KUKA KRL program: MyProgram_177().src

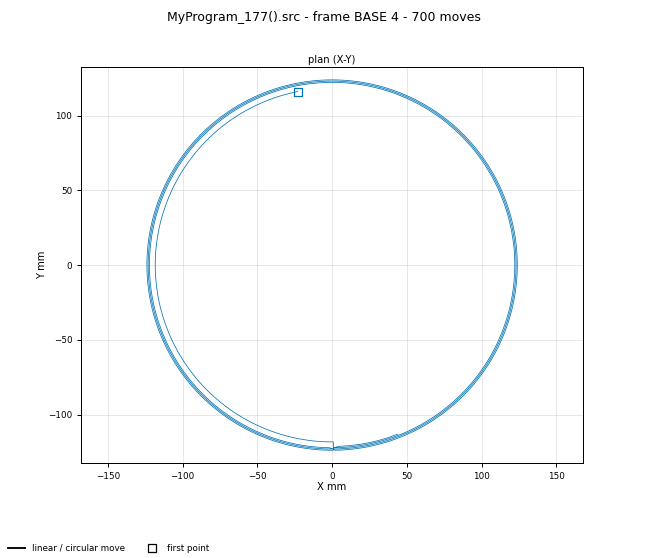
[picture p0: tool path of MyProgram_177().src in frame BASE 4, 700 of 700 moves have a stored position in this frame; points joined in program order, loops and branches not executed]
&ACCESS RVP
&REL 1
&PARAM TEMPLATE = C:\KRC\Roboter\Template\vorgabe
&PARAM EDITMASK = *
DEF MyProgram_177()
; ---- Setting reference (Base) ----
$BASE = BASE_DATA[4]

; --------------------------
; ---- Setting tool (TCP) ----
$TOOL = TOOL_DATA[3]
; --------------------------

$VEL.CP = VEL_APROX_PRINT
Startdeposition()
$VEL.CP = VEL_PRINT
LIN {X -23.0554,Y 116.0381,Z 130,A 97.2473,B 24.9369,C -1.8336,E1 24.968,E2 348.7277} C_DIS
LIN {X -25.5832,Y 115.5056,Z 130,A 98.5297,B 24.9369,C -1.8339,E1 24.9645,E2 347.4431} C_DIS
LIN {X -28.4099,Y 114.843,Z 130,A 99.9093,B 24.9371,C -1.8314,E1 24.9608,E2 346.0675} C_DIS
LIN {X -31.5451,Y 114.0233,Z 130,A 101.4825,B 24.9372,C -1.8299,E1 24.9566,E2 344.4954} C_DIS
LIN {X -33.9988,Y 113.3142,Z 130,A 102.7524,B 24.9372,C -1.8299,E1 24.9532,E2 343.2232} C_DIS
LIN {X -38.179,Y 111.9751,Z 130,A 104.8537,B 24.9375,C -1.8263,E1 24.9476,E2 341.1266} C_DIS
LIN {X -41.2308,Y 110.8892,Z 130,A 106.4224,B 24.9376,C -1.8243,E1 24.9435,E2 339.5598} C_DIS
LIN {X -43.9338,Y 109.8464,Z 130,A 107.833,B 24.9377,C -1.8227,E1 24.9398,E2 338.1499} C_DIS
LIN {X -46.5663,Y 108.7563,Z 130,A 109.2196,B 24.9378,C -1.8209,E1 24.9363,E2 336.7642} C_DIS
LIN {X -48.9465,Y 107.7046,Z 130,A 110.5124,B 24.9378,C -1.8205,E1 24.933,E2 335.4694} C_DIS
LIN {X -51.8783,Y 106.3252,Z 130,A 112.0577,B 24.9381,C -1.8169,E1 24.9291,E2 333.9286} C_DIS
LIN {X -54.4655,Y 105.0233,Z 130,A 113.4668,B 24.9383,C -1.8149,E1 24.9256,E2 332.5205} C_DIS
LIN {X -56.7349,Y 103.8132,Z 130,A 114.744,B 24.9383,C -1.8141,E1 24.9224,E2 331.2415} C_DIS
LIN {X -59.5311,Y 102.237,Z 130,A 116.2695,B 24.9386,C -1.81,E1 24.9188,E2 329.7212} C_DIS
LIN {X -61.9831,Y 100.769,Z 130,A 117.6521,B 24.9388,C -1.8074,E1 24.9155,E2 328.3406} C_DIS
LIN {X -64.0841,Y 99.4443,Z 130,A 118.8954,B 24.9388,C -1.8069,E1 24.9125,E2 327.0945} C_DIS
LIN {X -66.9275,Y 97.5557,Z 130,A 120.5341,B 24.9391,C -1.8029,E1 24.9087,E2 325.4598} C_DIS
LIN {X -69.0267,Y 96.0799,Z 130,A 121.7828,B 24.9392,C -1.8006,E1 24.9059,E2 324.2122} C_DIS
LIN {X -71.633,Y 94.1548,Z 130,A 123.5319,B 24.9389,C -1.805,E1 24.902,E2 322.4465} C_DIS
LIN {X -74.471,Y 91.9237,Z 130,A 125.1574,B 24.9395,C -1.7959,E1 24.8985,E2 320.8364} C_DIS
LIN {X -77.1406,Y 89.6968,Z 130,A 126.8154,B 24.9399,C -1.791,E1 24.8949,E2 319.1838} C_DIS
LIN {X -79.8507,Y 87.2914,Z 130,A 128.6126,B 24.94,C -1.7887,E1 24.8912,E2 317.3847} C_DIS
LIN {X -82.1926,Y 85.0898,Z 130,A 130.1847,B 24.9402,C -1.7857,E1 24.888,E2 315.8135} C_DIS
LIN {X -84.4552,Y 82.8455,Z 130,A 131.7119,B 24.9405,C -1.7812,E1 24.885,E2 314.2906} C_DIS
LIN {X -87.0481,Y 80.1159,Z 130,A 133.5624,B 24.9408,C -1.7777,E1 24.8815,E2 312.4401} C_DIS
LIN {X -89.1013,Y 77.8257,Z 130,A 135.0151,B 24.9411,C -1.7723,E1 24.8788,E2 310.9937} C_DIS
LIN {X -90.9628,Y 75.6417,Z 130,A 136.4115,B 24.9414,C -1.769,E1 24.8763,E2 309.599} C_DIS
LIN {X -92.9224,Y 73.2212,Z 130,A 137.984,B 24.9414,C -1.7676,E1 24.8736,E2 308.0222} C_DIS
LIN {X -94.8616,Y 70.6921,Z 130,A 139.5059,B 24.9418,C -1.7625,E1 24.871,E2 306.5053} C_DIS
LIN {X -96.5243,Y 68.404,Z 130,A 140.8635,B 24.9421,C -1.7582,E1 24.8688,E2 305.1514} C_DIS
LIN {X -98.1662,Y 66.0259,Z 130,A 142.3018,B 24.9422,C -1.7559,E1 24.8665,E2 303.7114} C_DIS
LIN {X -99.6639,Y 63.742,Z 130,A 143.669,B 24.9423,C -1.754,E1 24.8645,E2 302.3418} C_DIS
LIN {X -101.2988,Y 61.1114,Z 130,A 145.1543,B 24.9427,C -1.749,E1 24.8623,E2 300.8607} C_DIS
LIN {X -102.7791,Y 58.5877,Z 130,A 146.5378,B 24.943,C -1.7435,E1 24.8604,E2 299.4833} C_DIS
LIN {X -104.342,Y 55.7598,Z 130,A 148.1086,B 24.9433,C -1.7391,E1 24.8583,E2 297.9147} C_DIS
LIN {X -105.5174,Y 53.4988,Z 130,A 149.3549,B 24.9435,C -1.7359,E1 24.8567,E2 296.6693} C_DIS
LIN {X -106.7928,Y 50.905,Z 130,A 150.7637,B 24.9438,C -1.732,E1 24.855,E2 295.2621} C_DIS
LIN {X -108.1446,Y 47.9701,Z 130,A 152.3355,B 24.9441,C -1.7275,E1 24.8532,E2 293.6924} C_DIS
LIN {X -109.0992,Y 45.7526,Z 130,A 153.4985,B 24.9443,C -1.7237,E1 24.8519,E2 292.5321} C_DIS
LIN {X -110.2525,Y 42.9001,Z 130,A 155.0459,B 24.9445,C -1.7214,E1 24.8503,E2 290.9814} C_DIS
LIN {X -111.2701,Y 40.1871,Z 130,A 156.4592,B 24.9447,C -1.7175,E1 24.849,E2 289.5696} C_DIS
LIN {X -112.3399,Y 37.0964,Z 130,A 158.0181,B 24.9451,C -1.7114,E1 24.8476,E2 288.0164} C_DIS
LIN {X -113.1108,Y 34.6696,Z 130,A 159.2945,B 24.9452,C -1.7093,E1 24.8465,E2 286.7375} C_DIS
LIN {X -113.9235,Y 31.8979,Z 130,A 160.6739,B 24.9456,C -1.704,E1 24.8455,E2 285.3627} C_DIS
LIN {X -114.6486,Y 29.1833,Z 130,A 162.0888,B 24.9457,C -1.7019,E1 24.8445,E2 283.9447} C_DIS
LIN {X -115.5988,Y 25.1558,Z 130,A 164.0727,B 24.9462,C -1.6946,E1 24.8432,E2 281.9665} C_DIS
LIN {X -116.2045,Y 22.1911,Z 130,A 165.6096,B 24.9462,C -1.6928,E1 24.8424,E2 280.4247} C_DIS
LIN {X -116.8055,Y 18.785,Z 130,A 167.2246,B 24.9468,C -1.6848,E1 24.8417,E2 278.8193} C_DIS
LIN {X -117.1691,Y 16.352,Z 130,A 168.4696,B 24.9469,C -1.6832,E1 24.8412,E2 277.5707} C_DIS
LIN {X -117.5452,Y 13.3852,Z 130,A 169.884,B 24.9473,C -1.6771,E1 24.8407,E2 276.1624} C_DIS
LIN {X -117.8037,Y 10.8709,Z 130,A 171.128,B 24.9475,C -1.6739,E1 24.8404,E2 274.9185} C_DIS
LIN {X -118.0453,Y 7.824,Z 130,A 172.6425,B 24.9477,C -1.6705,E1 24.8401,E2 273.4031} C_DIS
LIN {X -118.2117,Y 4.6949,Z 130,A 174.1647,B 24.948,C -1.6657,E1 24.8399,E2 271.8831} C_DIS
LIN {X -118.2975,Y 1.4546,Z 130,A 175.7155,B 24.9484,C -1.6597,E1 24.8398,E2 270.3372} C_DIS
LIN {X -118.2771,Y -2.5603,Z 130,A 177.6649,B 24.9488,C -1.6536,E1 24.8398,E2 268.3906} C_DIS
LIN {X -118.1636,Y -5.8118,Z 130,A 179.26,B 24.949,C -1.6493,E1 24.84,E2 266.7962} C_DIS
LIN {X -118.0091,Y -8.3599,Z 130,A -179.4931,B 24.9492,C -1.6457,E1 24.8403,E2 265.5503} C_DIS
LIN {X -117.7689,Y -11.248,Z 130,A -178.1014,B 24.9496,C -1.6407,E1 24.8406,E2 264.1622} C_DIS
LIN {X -117.4472,Y -14.2216,Z 130,A -176.6275,B 24.9498,C -1.6371,E1 24.8411,E2 262.6881} C_DIS
LIN {X -117.0254,Y -17.363,Z 130,A -175.0769,B 24.95,C -1.6328,E1 24.8417,E2 261.1385} C_DIS
LIN {X -116.6213,Y -19.8875,Z 130,A -173.8288,B 24.9503,C -1.6293,E1 24.8423,E2 259.8914} C_DIS
LIN {X -116.034,Y -23.0767,Z 130,A -172.2471,B 24.9505,C -1.6248,E1 24.8431,E2 258.3111} C_DIS
LIN {X -115.5071,Y -25.5762,Z 130,A -170.97,B 24.9507,C -1.6226,E1 24.8438,E2 257.0317} C_DIS
LIN {X -114.8418,Y -28.4149,Z 130,A -169.5763,B 24.951,C -1.6174,E1 24.8448,E2 255.6422} C_DIS
LIN {X -114.0131,Y -31.5816,Z 130,A -167.9878,B 24.9513,C -1.6126,E1 24.8459,E2 254.0559} C_DIS
LIN {X -113.3057,Y -34.0276,Z 130,A -166.7136,B 24.9513,C -1.6106,E1 24.8469,E2 252.7791} C_DIS
LIN {X -112.3496,Y -37.0666,Z 130,A -165.1953,B 24.9517,C -1.6048,E1 24.8482,E2 251.2658} C_DIS
LIN {X -111.5091,Y -39.5191,Z 130,A -163.8965,B 24.9519,C -1.6029,E1 24.8494,E2 249.9643} C_DIS
LIN {X -110.5112,Y -42.2291,Z 130,A -162.511,B 24.9521,C -1.5982,E1 24.8508,E2 248.5823} C_DIS
LIN {X -109.4666,Y -44.8668,Z 130,A -161.0898,B 24.9523,C -1.5961,E1 24.8523,E2 247.158} C_DIS
LIN {X -108.1572,Y -47.9419,Z 130,A -159.5069,B 24.9526,C -1.5899,E1 24.854,E2 245.5813} C_DIS
LIN {X -106.9506,Y -50.5764,Z 130,A -158.0948,B 24.9529,C -1.5862,E1 24.8557,E2 244.1702} C_DIS
LIN {X -105.8441,Y -52.8491,Z 130,A -156.831,B 24.9529,C -1.5845,E1 24.8572,E2 242.9037} C_DIS
LIN {X -104.3807,Y -55.6863,Z 130,A -155.3234,B 24.9533,C -1.5785,E1 24.8592,E2 241.4023} C_DIS
LIN {X -103.0732,Y -58.069,Z 130,A -154.0102,B 24.9535,C -1.5748,E1 24.861,E2 240.0911} C_DIS
LIN {X -101.4733,Y -60.8242,Z 130,A -152.4327,B 24.9537,C -1.572,E1 24.8632,E2 238.512} C_DIS
LIN {X -100.1359,Y -62.9987,Z 130,A -151.1882,B 24.9539,C -1.5691,E1 24.8651,E2 237.268} C_DIS
LIN {X -98.5628,Y -65.4325,Z 130,A -149.7472,B 24.9539,C -1.5671,E1 24.8673,E2 235.8247} C_DIS
LIN {X -96.7218,Y -68.1271,Z 130,A -148.1903,B 24.9543,C -1.562,E1 24.8697,E2 234.2722} C_DIS
LIN {X -95.2246,Y -70.2019,Z 130,A -146.9154,B 24.9543,C -1.5604,E1 24.8718,E2 232.9948} C_DIS
LIN {X -92.9467,Y -73.1904,Z 130,A -145.068,B 24.9546,C -1.5572,E1 24.875,E2 231.1465} C_DIS
LIN {X -90.8987,Y -75.7188,Z 130,A -143.4713,B 24.9547,C -1.5543,E1 24.8778,E2 229.5491} C_DIS
LIN {X -88.6316,Y -78.3636,Z 130,A -141.6581,B 24.9547,C -1.5558,E1 24.8812,E2 227.7242} C_DIS
LIN {X -86.1773,Y -81.0516,Z 130,A -140.0286,B 24.9552,C -1.5461,E1 24.8842,E2 226.1106} C_DIS
LIN {X -83.7815,Y -83.5275,Z 130,A -138.385,B 24.9555,C -1.5414,E1 24.8875,E2 224.4712} C_DIS
LIN {X -81.7148,Y -85.5504,Z 130,A -136.8233,B 24.9553,C -1.5454,E1 24.8906,E2 222.8935} C_DIS
LIN {X -78.9462,Y -88.1102,Z 130,A -135.1327,B 24.9558,C -1.5359,E1 24.8941,E2 221.2188} C_DIS
LIN {X -76.7251,Y -90.0508,Z 130,A -133.7096,B 24.956,C -1.5328,E1 24.8971,E2 219.7974} C_DIS
LIN {X -74.4958,Y -91.9036,Z 130,A -132.266,B 24.956,C -1.5319,E1 24.9002,E2 218.3505} C_DIS
LIN {X -71.882,Y -93.963,Z 130,A -130.6607,B 24.9562,C -1.5287,E1 24.9038,E2 216.7471} C_DIS
LIN {X -69.3743,Y -95.8306,Z 130,A -129.1752,B 24.9564,C -1.5247,E1 24.9071,E2 215.2656} C_DIS
LIN {X -67.3753,Y -97.2445,Z 130,A -127.9426,B 24.9564,C -1.5248,E1 24.9099,E2 214.0286} C_DIS
LIN {X -64.5186,Y -99.1654,Z 130,A -126.2982,B 24.9567,C -1.5211,E1 24.9137,E2 212.3877} C_DIS
LIN {X -62.0717,Y -100.715,Z 130,A -124.8924,B 24.9567,C -1.5191,E1 24.9171,E2 210.9822} C_DIS
LIN {X -59.5882,Y -102.2039,Z 130,A -123.4898,B 24.9569,C -1.517,E1 24.9204,E2 209.5803} C_DIS
LIN {X -56.3394,Y -104.0278,Z 130,A -121.6241,B 24.9569,C -1.5173,E1 24.925,E2 207.7086} C_DIS
LIN {X -53.4928,Y -105.5204,Z 130,A -120.1136,B 24.9571,C -1.5132,E1 24.9288,E2 206.2036} C_DIS
LIN {X -50.8925,Y -106.7988,Z 130,A -118.7067,B 24.9571,C -1.5117,E1 24.9323,E2 204.7968} C_DIS
LIN {X -47.9481,Y -108.1545,Z 130,A -117.1334,B 24.9573,C -1.51,E1 24.9363,E2 203.2237} C_DIS
LIN {X -45.5917,Y -109.167,Z 130,A -115.8881,B 24.9573,C -1.5088,E1 24.9395,E2 201.9782} C_DIS
LIN {X -42.9107,Y -110.2483,Z 130,A -114.4552,B 24.9573,C -1.5089,E1 24.9432,E2 200.542} C_DIS
LIN {X -40.3374,Y -111.2152,Z 130,A -113.0897,B 24.9573,C -1.5092,E1 24.9468,E2 199.1729} C_DIS
LIN {X -37.1077,Y -112.3362,Z 130,A -111.4933,B 24.9576,C -1.5052,E1 24.951,E2 197.5832} C_DIS
LIN {X -34.6731,Y -113.1097,Z 130,A -110.224,B 24.9576,C -1.5057,E1 24.9544,E2 196.3103} C_DIS
LIN {X -30.7346,Y -114.2422,Z 130,A -108.2401,B 24.9576,C -1.5044,E1 24.9597,E2 194.3265} C_DIS
LIN {X -27.3386,Y -115.1044,Z 130,A -106.5664,B 24.9577,C -1.5023,E1 24.9643,E2 192.6553} C_DIS
LIN {X -24.4991,Y -115.742,Z 130,A -105.1569,B 24.9577,C -1.5017,E1 24.9681,E2 191.2456} C_DIS
LIN {X -21.9964,Y -116.242,Z 130,A -103.8895,B 24.9577,C -1.5027,E1 24.9716,E2 189.9745} C_DIS
LIN {X -18.8077,Y -116.8018,Z 130,A -102.3491,B 24.9577,C -1.5009,E1 24.9758,E2 188.4369} C_DIS
LIN {X -16.2845,Y -117.1786,Z 130,A -101.0828,B 24.9577,C -1.502,E1 24.9794,E2 187.1668} C_DIS
LIN {X -13.4152,Y -117.5417,Z 130,A -99.7079,B 24.9578,C -1.5006,E1 24.9832,E2 185.7943} C_DIS
LIN {X -10.1586,Y -117.8695,Z 130,A -98.1265,B 24.9578,C -1.5003,E1 24.9876,E2 184.2128} C_DIS
LIN {X -7.2772,Y -118.0823,Z 130,A -96.7302,B 24.9578,C -1.5002,E1 24.9914,E2 182.8163} C_DIS
LIN {X -4.7355,Y -118.2099,Z 130,A -95.4636,B 24.9578,C -1.5019,E1 24.995,E2 181.5455} C_DIS
LIN {X -1.5126,Y -118.2964,Z 130,A -93.9402,B 24.9578,C -1.5004,E1 24.9992,E2 180.0255} C_DIS
LIN {X 0.8051,Y -118.3,Z 130,A -93.2857,B 24.959,C -1.4793,E1 25.0009,E2 179.4209} C_DIS
Enddeposition()
LIN {X 0.8803,Y -123.8691,Z 131,A -92.8411,B 24.9628,C -1.4093,E1 25.0017,E2 179.1423} C_DIS
Startdeposition()
$VEL.CP = VEL_PRINT
LIN {X -2.0906,Y -123.8586,Z 131,A -94.6443,B 24.9639,C -1.3883,E1 24.9965,E2 180.9953} C_DIS
LIN {X -5.7833,Y -123.7415,Z 131,A -96.4357,B 24.9641,C -1.3841,E1 24.9915,E2 182.7968} C_DIS
LIN {X -9.9561,Y -123.475,Z 131,A -98.2533,B 24.9638,C -1.3897,E1 24.9865,E2 184.602} C_DIS
LIN {X -13.6339,Y -123.1241,Z 131,A -100.013,B 24.9639,C -1.3874,E1 24.9816,E2 186.3681} C_DIS
LIN {X -17.2995,Y -122.6617,Z 131,A -101.7668,B 24.964,C -1.3857,E1 24.9767,E2 188.1273} C_DIS
LIN {X -21.4294,Y -122.009,Z 131,A -103.7033,B 24.964,C -1.3861,E1 24.9714,E2 190.0645} C_DIS
LIN {X -25.0583,Y -121.3152,Z 131,A -105.4226,B 24.964,C -1.3863,E1 24.9666,E2 191.7853} C_DIS
LIN {X -29.1383,Y -120.4006,Z 131,A -107.2922,B 24.9638,C -1.3904,E1 24.9616,E2 193.6478} C_DIS
LIN {X -32.7159,Y -119.4783,Z 131,A -109.0799,B 24.9639,C -1.3877,E1 24.9567,E2 195.4445} C_DIS
LIN {X -36.7293,Y -118.3054,Z 131,A -110.9071,B 24.9636,C -1.3941,E1 24.9519,E2 197.2596} C_DIS
LIN {X -40.2412,Y -117.1583,Z 131,A -112.7389,B 24.9638,C -1.3898,E1 24.947,E2 199.1052} C_DIS
LIN {X -43.7167,Y -115.9051,Z 131,A -114.4193,B 24.9637,C -1.3927,E1 24.9426,E2 200.7821} C_DIS
LIN {X -47.6039,Y -114.3647,Z 131,A -116.3998,B 24.9637,C -1.3925,E1 24.9375,E2 202.7674} C_DIS
LIN {X -50.993,Y -112.8938,Z 131,A -118.0807,B 24.9635,C -1.3957,E1 24.9332,E2 204.4448} C_DIS
LIN {X -54.0022,Y -111.4861,Z 131,A -119.6317,B 24.9635,C -1.3968,E1 24.9293,E2 205.9969} C_DIS
LIN {X -57.7337,Y -109.5995,Z 131,A -121.4661,B 24.9631,C -1.404,E1 24.9247,E2 207.8195} C_DIS
LIN {X -60.9768,Y -107.8297,Z 131,A -123.1166,B 24.9628,C -1.409,E1 24.9207,E2 209.4627} C_DIS
LIN {X -63.8464,Y -106.1558,Z 131,A -124.847,B 24.9632,C -1.4023,E1 24.9165,E2 211.2142} C_DIS
LIN {X -67.3976,Y -103.9363,Z 131,A -126.7652,B 24.963,C -1.4063,E1 24.912,E2 213.1292} C_DIS
LIN {X -70.768,Y -101.6719,Z 131,A -128.6431,B 24.9628,C -1.4094,E1 24.9077,E2 215.006} C_DIS
LIN {X -73.4693,Y -99.7379,Z 131,A -130.1959,B 24.9627,C -1.4113,E1 24.9042,E2 216.5596} C_DIS
LIN {X -76.7931,Y -97.2012,Z 131,A -132.0376,B 24.9623,C -1.419,E1 24.9001,E2 218.3897} C_DIS
LIN {X -79.6581,Y -94.8684,Z 131,A -133.6869,B 24.962,C -1.425,E1 24.8966,E2 220.0311} C_DIS
LIN {X -82.1734,Y -92.6982,Z 131,A -135.4172,B 24.9623,C -1.4193,E1 24.8929,E2 221.7818} C_DIS
LIN {X -84.9008,Y -90.2059,Z 131,A -137.1015,B 24.962,C -1.4239,E1 24.8895,E2 223.462} C_DIS
LIN {X -87.8971,Y -87.2896,Z 131,A -139.0407,B 24.9618,C -1.4278,E1 24.8856,E2 225.4} C_DIS
LIN {X -90.4611,Y -84.6295,Z 131,A -140.7717,B 24.9617,C -1.4306,E1 24.8823,E2 227.1319} C_DIS
LIN {X -93.2654,Y -81.5281,Z 131,A -142.6207,B 24.9612,C -1.4389,E1 24.8789,E2 228.9695} C_DIS
LIN {X -95.4176,Y -78.9974,Z 131,A -144.1308,B 24.961,C -1.4437,E1 24.8762,E2 230.475} C_DIS
LIN {X -97.732,Y -76.1175,Z 131,A -145.998,B 24.9611,C -1.4407,E1 24.8729,E2 232.3581} C_DIS
LIN {X -99.9579,Y -73.1688,Z 131,A -147.6386,B 24.9607,C -1.4481,E1 24.8702,E2 233.9891} C_DIS
LIN {X -101.8844,Y -70.4622,Z 131,A -149.2395,B 24.9607,C -1.4491,E1 24.8676,E2 235.5954} C_DIS
LIN {X -104.2041,Y -66.9834,Z 131,A -151.0939,B 24.9602,C -1.4577,E1 24.8648,E2 237.4386} C_DIS
LIN {X -105.9624,Y -64.1647,Z 131,A -152.605,B 24.9599,C -1.463,E1 24.8626,E2 238.945} C_DIS
LIN {X -107.8297,Y -60.9768,Z 131,A -154.4692,B 24.96,C -1.4607,E1 24.86,E2 240.8243} C_DIS
LIN {X -109.5995,Y -57.7337,Z 131,A -156.1081,B 24.9596,C -1.4686,E1 24.8578,E2 242.4532} C_DIS
LIN {X -111.1087,Y -54.7741,Z 131,A -157.7126,B 24.9596,C -1.4699,E1 24.8558,E2 244.0631} C_DIS
LIN {X -112.8938,Y -50.993,Z 131,A -159.5726,B 24.959,C -1.4787,E1 24.8536,E2 245.9122} C_DIS
LIN {X -114.3647,Y -47.6039,Z 131,A -161.3885,B 24.959,C -1.479,E1 24.8516,E2 247.7375} C_DIS
LIN {X -115.7823,Y -44.0402,Z 131,A -163.1137,B 24.9586,C -1.4864,E1 24.8499,E2 249.4547} C_DIS
LIN {X -117.1299,Y -40.3226,Z 131,A -165.034,B 24.9586,C -1.4879,E1 24.8481,E2 251.3824} C_DIS
LIN {X -118.3054,Y -36.7293,Z 131,A -166.7528,B 24.9582,C -1.4946,E1 24.8467,E2 253.0952} C_DIS
LIN {X -119.4783,Y -32.7159,Z 131,A -168.7073,B 24.9579,C -1.4996,E1 24.8452,E2 255.0489} C_DIS
LIN {X -120.4006,Y -29.1383,Z 131,A -170.4303,B 24.9576,C -1.5043,E1 24.844,E2 256.7708} C_DIS
LIN {X -121.3152,Y -25.0583,Z 131,A -172.2977,B 24.9571,C -1.5134,E1 24.8429,E2 258.6276} C_DIS
LIN {X -122.009,Y -21.4294,Z 131,A -174.1081,B 24.9571,C -1.5143,E1 24.842,E2 260.4465} C_DIS
LIN {X -122.6617,Y -17.2995,Z 131,A -175.9319,B 24.9564,C -1.5254,E1 24.8412,E2 262.2548} C_DIS
LIN {X -123.1241,Y -13.6339,Z 131,A -177.7864,B 24.9564,C -1.5245,E1 24.8406,E2 264.1225} C_DIS
LIN {X -123.4741,Y -9.9669,Z 131,A -179.4725,B 24.9561,C -1.5308,E1 24.8402,E2 265.8037} C_DIS
LIN {X -123.7415,Y -5.7833,Z 131,A 178.535,B 24.9559,C -1.5348,E1 24.8399,E2 267.7988} C_DIS
LIN {X -123.8586,Y -2.0906,Z 131,A 176.8453,B 24.9555,C -1.5412,E1 24.8398,E2 269.4833} C_DIS
LIN {X -123.8644,Y 1.6717,Z 131,A 175.0982,B 24.9552,C -1.5466,E1 24.8398,E2 271.228} C_DIS
LIN {X -123.7415,Y 5.7833,Z 131,A 173.1675,B 24.9549,C -1.5516,E1 24.84,E2 273.1585} C_DIS
LIN {X -123.475,Y 9.9561,Z 131,A 171.3372,B 24.9543,C -1.5625,E1 24.8404,E2 274.9738} C_DIS
LIN {X -123.1241,Y 13.6339,Z 131,A 169.4888,B 24.9543,C -1.5619,E1 24.8409,E2 276.8345} C_DIS
LIN {X -122.6617,Y 17.2995,Z 131,A 167.8051,B 24.9539,C -1.5686,E1 24.8415,E2 278.5123} C_DIS
LIN {X -122.009,Y 21.4294,Z 131,A 165.8101,B 24.9537,C -1.5723,E1 24.8425,E2 280.5105} C_DIS
LIN {X -121.3152,Y 25.0583,Z 131,A 164.1215,B 24.9533,C -1.5787,E1 24.8434,E2 282.1937} C_DIS
LIN {X -120.4006,Y 29.1383,Z 131,A 162.2411,B 24.9528,C -1.5873,E1 24.8446,E2 284.0647} C_DIS
LIN {X -119.4783,Y 32.7159,Z 131,A 160.4433,B 24.9527,C -1.5889,E1 24.8458,E2 285.8692} C_DIS
LIN {X -118.3054,Y 36.7293,Z 131,A 158.6065,B 24.9521,C -1.5993,E1 24.8473,E2 287.6917} C_DIS
LIN {X -117.1583,Y 40.2412,Z 131,A 156.7653,B 24.9521,C -1.599,E1 24.849,E2 289.5443} C_DIS
LIN {X -115.9051,Y 43.7167,Z 131,A 155.0769,B 24.9517,C -1.6052,E1 24.8506,E2 291.2273} C_DIS
LIN {X -114.3647,Y 47.6039,Z 131,A 153.0875,B 24.9515,C -1.6088,E1 24.8527,E2 293.2193} C_DIS
LIN {X -112.8938,Y 50.993,Z 131,A 151.3995,B 24.9511,C -1.615,E1 24.8546,E2 294.9018} C_DIS
LIN {X -111.4861,Y 54.0022,Z 131,A 149.8425,B 24.9509,C -1.6187,E1 24.8565,E2 296.4584} C_DIS
LIN {X -109.5995,Y 57.7337,Z 131,A 148.0014,B 24.9503,C -1.6286,E1 24.8588,E2 298.2857} C_DIS
LIN {X -107.8297,Y 60.9768,Z 131,A 146.3455,B 24.9498,C -1.636,E1 24.861,E2 299.9328} C_DIS
LIN {X -106.1558,Y 63.8464,Z 131,A 144.6093,B 24.9501,C -1.6317,E1 24.8635,E2 301.6881} C_DIS
LIN {X -104.2041,Y 66.9834,Z 131,A 142.922,B 24.9498,C -1.6376,E1 24.866,E2 303.37} C_DIS
LIN {X -102.3707,Y 69.7539,Z 131,A 141.3656,B 24.9495,C -1.641,E1 24.8684,E2 304.9259} C_DIS
LIN {X -99.9579,Y 73.1688,Z 131,A 139.5211,B 24.949,C -1.6504,E1 24.8714,E2 306.7573} C_DIS
LIN {X -97.732,Y 76.1175,Z 131,A 137.8709,B 24.9485,C -1.6576,E1 24.8742,E2 308.3981} C_DIS
LIN {X -95.6678,Y 78.696,Z 131,A 136.1502,B 24.9488,C -1.6531,E1 24.8773,E2 310.1374} C_DIS
LIN {X -93.2654,Y 81.5281,Z 131,A 134.4487,B 24.9485,C -1.6583,E1 24.8804,E2 311.8342} C_DIS
LIN {X -91.0459,Y 84.0001,Z 131,A 132.8932,B 24.9483,C -1.6614,E1 24.8833,E2 313.3893} C_DIS
LIN {X -88.2958,Y 86.8851,Z 131,A 131.1065,B 24.9478,C -1.6685,E1 24.8867,E2 315.1667} C_DIS
LIN {X -85.793,Y 89.357,Z 131,A 129.5354,B 24.9474,C -1.675,E1 24.8899,E2 316.7291} C_DIS
LIN {X -83.091,Y 91.8766,Z 131,A 127.6663,B 24.9476,C -1.6719,E1 24.8937,E2 318.6132} C_DIS
LIN {X -80.3137,Y 94.3131,Z 131,A 126.025,B 24.9472,C -1.6788,E1 24.8972,E2 320.2444} C_DIS
LIN {X -77.7559,Y 96.4333,Z 131,A 124.4266,B 24.9472,C -1.6794,E1 24.9006,E2 321.8473} C_DIS
LIN {X -74.4569,Y 99.0022,Z 131,A 122.5761,B 24.9466,C -1.6873,E1 24.9047,E2 323.6858} C_DIS
LIN {X -71.7749,Y 100.9628,Z 131,A 121.0669,B 24.9464,C -1.6917,E1 24.9081,E2 325.1897} C_DIS
LIN {X -68.7329,Y 103.0593,Z 131,A 119.2034,B 24.9466,C -1.6882,E1 24.9125,E2 327.0679} C_DIS
LIN {X -65.6285,Y 105.0625,Z 131,A 117.5662,B 24.9462,C -1.6947,E1 24.9163,E2 328.6948} C_DIS
LIN {X -62.8455,Y 106.7509,Z 131,A 115.9864,B 24.9462,C -1.6942,E1 24.9201,E2 330.2807} C_DIS
LIN {X -59.1894,Y 108.8204,Z 131,A 114.1294,B 24.9457,C -1.7015,E1 24.9246,E2 332.1258} C_DIS
LIN {X -56.2077,Y 110.3894,Z 131,A 112.6052,B 24.9455,C -1.7056,E1 24.9284,E2 333.6442} C_DIS
LIN {X -52.8913,Y 112.0176,Z 131,A 110.7476,B 24.9457,C -1.7016,E1 24.9331,E2 335.5161} C_DIS
LIN {X -49.5269,Y 113.5443,Z 131,A 109.0771,B 24.9455,C -1.706,E1 24.9373,E2 337.1803} C_DIS
LIN {X -45.667,Y 115.1517,Z 131,A 107.0831,B 24.9455,C -1.706,E1 24.9425,E2 339.1787} C_DIS
LIN {X -42.2126,Y 116.4622,Z 131,A 105.4014,B 24.9452,C -1.7094,E1 24.9469,E2 340.8556} C_DIS
LIN {X -38.2581,Y 117.8203,Z 131,A 103.5452,B 24.9449,C -1.7154,E1 24.9518,E2 342.7013} C_DIS
LIN {X -34.7276,Y 118.9092,Z 131,A 101.7391,B 24.945,C -1.7128,E1 24.9566,E2 344.5164} C_DIS
LIN {X -30.6946,Y 120.0125,Z 131,A 99.9271,B 24.9445,C -1.7204,E1 24.9615,E2 346.3131} C_DIS
LIN {X -27.1022,Y 120.8755,Z 131,A 98.0785,B 24.9448,C -1.7156,E1 24.9665,E2 348.1756} C_DIS
LIN {X -23.4853,Y 121.6291,Z 131,A 96.3986,B 24.9447,C -1.7184,E1 24.9711,E2 349.8509} C_DIS
LIN {X -19.3673,Y 122.3532,Z 131,A 94.4194,B 24.9447,C -1.7177,E1 24.9766,E2 351.8336} C_DIS
LIN {X -15.7099,Y 122.8761,Z 131,A 92.7402,B 24.9445,C -1.7201,E1 24.9812,E2 353.5082} C_DIS
LIN {X -11.554,Y 123.3362,Z 131,A 90.88,B 24.9443,C -1.7246,E1 24.9864,E2 355.3589} C_DIS
LIN {X -7.8709,Y 123.6263,Z 131,A 89.0835,B 24.9445,C -1.7212,E1 24.9914,E2 357.1641} C_DIS
LIN {X -4.0407,Y 123.8094,Z 131,A 87.3613,B 24.9443,C -1.7242,E1 24.9962,E2 358.8796} C_DIS
LIN {X 0,Y 123.8767,Z 131,A 85.4283,B 24.9445,C -1.7217,E1 25.0016,E2 360.8186} C_DIS
LIN {X 3.6941,Y 123.8206,Z 131,A 83.7509,B 24.9443,C -1.7233,E1 25.0063,E2 362.4918} C_DIS
LIN {X 7.8709,Y 123.6263,Z 131,A 81.7746,B 24.9445,C -1.7214,E1 25.0118,E2 364.472} C_DIS
LIN {X 11.554,Y 123.3362,Z 131,A 80.098,B 24.9444,C -1.7227,E1 25.0164,E2 366.1444} C_DIS
LIN {X 15.7099,Y 122.8761,Z 131,A 78.2344,B 24.9442,C -1.7257,E1 25.0216,E2 367.9997} C_DIS
LIN {X 19.3673,Y 122.3532,Z 131,A 76.4468,B 24.9445,C -1.7215,E1 25.0265,E2 369.7956} C_DIS
LIN {X 23.4853,Y 121.6291,Z 131,A 74.6276,B 24.9442,C -1.7261,E1 25.0315,E2 371.6017} C_DIS
LIN {X 27.1022,Y 120.8755,Z 131,A 72.7973,B 24.9446,C -1.7195,E1 25.0365,E2 373.4453} C_DIS
LIN {X 30.6946,Y 120.0125,Z 131,A 71.1223,B 24.9446,C -1.7201,E1 25.0411,E2 375.1164} C_DIS
LIN {X 34.7276,Y 118.9092,Z 131,A 69.1492,B 24.9448,C -1.7169,E1 25.0464,E2 377.0939} C_DIS
LIN {X 38.2581,Y 117.8203,Z 131,A 67.4752,B 24.9448,C -1.7172,E1 25.0508,E2 378.7641} C_DIS
LIN {X 41.9066,Y 116.572,Z 131,A 65.7118,B 24.9448,C -1.7166,E1 25.0555,E2 380.5254} C_DIS
LIN {X 45.667,Y 115.1517,Z 131,A 63.8296,B 24.945,C -1.7136,E1 25.0604,E2 382.4105} C_DIS
LIN {X 49.5269,Y 113.5443,Z 131,A 62.0067,B 24.9448,C -1.7168,E1 25.065,E2 384.2215} C_DIS
LIN {X 52.8913,Y 112.0176,Z 131,A 60.3639,B 24.9447,C -1.718,E1 25.0692,E2 385.8574} C_DIS
LIN {X 55.8761,Y 110.5589,Z 131,A 58.6427,B 24.9454,C -1.7071,E1 25.0735,E2 387.5998} C_DIS
LIN {X 59.148,Y 108.843,Z 131,A 56.9705,B 24.9454,C -1.7065,E1 25.0776,E2 389.2685} C_DIS
LIN {X 62.0457,Y 107.218,Z 131,A 55.4284,B 24.9456,C -1.704,E1 25.0814,E2 390.8119} C_DIS
LIN {X 65.6285,Y 105.0625,Z 131,A 53.6027,B 24.9454,C -1.7063,E1 25.0857,E2 392.6264} C_DIS
LIN {X 68.7329,Y 103.0593,Z 131,A 51.9643,B 24.9454,C -1.707,E1 25.0895,E2 394.2579} C_DIS
LIN {X 71.4718,Y 101.1791,Z 131,A 50.2461,B 24.9461,C -1.6955,E1 25.0935,E2 395.9973} C_DIS
LIN {X 74.4569,Y 99.0022,Z 131,A 48.5756,B 24.9462,C -1.6943,E1 25.0973,E2 397.6646} C_DIS
LIN {X 77.0853,Y 96.9703,Z 131,A 47.0347,B 24.9464,C -1.6912,E1 25.1006,E2 399.2071} C_DIS
LIN {X 80.1972,Y 94.4118,Z 131,A 45.2544,B 24.9464,C -1.6917,E1 25.1044,E2 400.9795} C_DIS
LIN {X 83.091,Y 91.8766,Z 131,A 43.5719,B 24.9463,C -1.6928,E1 25.1079,E2 402.6526} C_DIS
LIN {X 85.5248,Y 89.6154,Z 131,A 41.8571,B 24.9471,C -1.6808,E1 25.1115,E2 404.3887} C_DIS
LIN {X 88.1588,Y 87.0246,Z 131,A 40.2299,B 24.9471,C -1.6811,E1 25.1147,E2 406.0082} C_DIS
LIN {X 90.4611,Y 84.6295,Z 131,A 38.648,B 24.9474,C -1.6755,E1 25.1177,E2 407.5967} C_DIS
LIN {X 93.1374,Y 81.6738,Z 131,A 36.8772,B 24.9474,C -1.6748,E1 25.121,E2 409.361} C_DIS
LIN {X 95.4176,Y 78.9974,Z 131,A 35.3221,B 24.9474,C -1.6745,E1 25.1238,E2 410.9097} C_DIS
LIN {X 97.732,Y 76.1175,Z 131,A 33.4741,B 24.9482,C -1.6634,E1 25.127,E2 412.7753} C_DIS
LIN {X 99.9579,Y 73.1688,Z 131,A 31.8061,B 24.9482,C -1.6612,E1 25.1298,E2 414.4406} C_DIS
LIN {X 102.4325,Y 69.6627,Z 131,A 29.8187,B 24.9486,C -1.6559,E1 25.133,E2 416.4307} C_DIS
LIN {X 104.4053,Y 66.67,Z 131,A 28.1734,B 24.9488,C -1.6522,E1 25.1355,E2 418.0766} C_DIS
LIN {X 106.5956,Y 63.1084,Z 131,A 26.3384,B 24.9488,C -1.6519,E1 25.1381,E2 419.9028} C_DIS
LIN {X 108.249,Y 60.2269,Z 131,A 24.8446,B 24.949,C -1.6498,E1 25.1401,E2 421.3937} C_DIS
LIN {X 109.998,Y 56.9725,Z 131,A 23.0035,B 24.9497,C -1.6384,E1 25.1426,E2 423.2521} C_DIS
LIN {X 111.6474,Y 53.6666,Z 131,A 21.3849,B 24.9497,C -1.6381,E1 25.1445,E2 424.8628} C_DIS
LIN {X 113.0468,Y 50.6535,Z 131,A 19.799,B 24.9501,C -1.6311,E1 25.1464,E2 426.4565} C_DIS
LIN {X 114.6917,Y 46.8094,Z 131,A 17.9611,B 24.9501,C -1.6303,E1 25.1484,E2 428.2863} C_DIS
LIN {X 116.037,Y 43.3685,Z 131,A 16.1691,B 24.9508,C -1.621,E1 25.1502,E2 430.0902} C_DIS
LIN {X 117.4336,Y 39.4273,Z 131,A 14.3743,B 24.9507,C -1.6222,E1 25.1518,E2 431.8722} C_DIS
LIN {X 118.5581,Y 35.9081,Z 131,A 12.5576,B 24.9513,C -1.6114,E1 25.1533,E2 433.7038} C_DIS
LIN {X 119.5754,Y 32.3564,Z 131,A 10.8736,B 24.9516,C -1.6074,E1 25.1546,E2 435.3876} C_DIS
LIN {X 120.6,Y 28.3026,Z 131,A 8.9106,B 24.952,C -1.5999,E1 25.1559,E2 437.357} C_DIS
LIN {X 121.3901,Y 24.6935,Z 131,A 7.2449,B 24.9522,C -1.5966,E1 25.1568,E2 439.0206} C_DIS
LIN {X 122.1543,Y 20.5827,Z 131,A 5.4014,B 24.9523,C -1.5951,E1 25.1577,E2 440.8571} C_DIS
LIN {X 122.7141,Y 16.9308,Z 131,A 3.6167,B 24.9529,C -1.5857,E1 25.1585,E2 442.6533} C_DIS
LIN {X 123.2147,Y 12.7796,Z 131,A 1.8166,B 24.9529,C -1.5863,E1 25.159,E2 444.4414} C_DIS
LIN {X 123.542,Y 9.0995,Z 131,A -0.0114,B 24.9535,C -1.5746,E1 25.1594,E2 446.286} C_DIS
LIN {X 123.7575,Y 5.4113,Z 131,A -1.6769,B 24.9537,C -1.5713,E1 25.1597,E2 447.9495} C_DIS
LIN {X 123.8704,Y 1.2315,Z 131,A -3.6412,B 24.9542,C -1.5634,E1 25.1597,E2 449.9207} C_DIS
LIN {X 123.832,Y -3.3219,Z 131,A -5.7303,B 24.9546,C -1.5573,E1 25.1597,E2 452.0116} C_DIS
LIN {X 123.6775,Y -7.0132,Z 131,A -7.3957,B 24.9548,C -1.5539,E1 25.1595,E2 453.6751} C_DIS
LIN {X 123.3704,Y -11.1832,Z 131,A -9.2462,B 24.9548,C -1.5518,E1 25.159,E2 455.5197} C_DIS
LIN {X 122.9823,Y -14.8573,Z 131,A -11.0235,B 24.9554,C -1.5427,E1 25.1585,E2 457.3079} C_DIS
LIN {X 122.4101,Y -18.9992,Z 131,A -12.8306,B 24.9554,C -1.5429,E1 25.1578,E2 459.104} C_DIS
LIN {X 121.79,Y -22.6414,Z 131,A -14.6512,B 24.9561,C -1.5316,E1 25.1569,E2 460.9405} C_DIS
LIN {X 121.0596,Y -26.263,Z 131,A -16.3166,B 24.9562,C -1.5282,E1 25.1559,E2 462.6042} C_DIS
LIN {X 120.1052,Y -30.3339,Z 131,A -18.2791,B 24.9567,C -1.5205,E1 25.1546,E2 464.5735} C_DIS
LIN {X 119.1468,Y -33.902,Z 131,A -19.9448,B 24.9569,C -1.5172,E1 25.1534,E2 466.2374} C_DIS
LIN {X 117.9349,Y -37.9038,Z 131,A -21.8016,B 24.957,C -1.5149,E1 25.1518,E2 468.089} C_DIS
LIN {X 116.7523,Y -41.4039,Z 131,A -23.5732,B 24.9575,C -1.5063,E1 25.1502,E2 469.8709} C_DIS
LIN {X 115.2879,Y -45.3203,Z 131,A -25.3872,B 24.9575,C -1.5063,E1 25.1484,E2 471.6748} C_DIS
LIN {X 113.8858,Y -48.7385,Z 131,A -27.0238,B 24.9575,C -1.5047,E1 25.1467,E2 473.3063} C_DIS
LIN {X 112.5378,Y -51.775,Z 131,A -28.7391,B 24.9584,C -1.4909,E1 25.1447,E2 475.0448} C_DIS
LIN {X 110.9433,Y -55.1078,Z 131,A -30.4051,B 24.9585,C -1.4879,E1 25.1426,E2 476.7091} C_DIS
LIN {X 109.426,Y -58.0632,Z 131,A -31.9423,B 24.9588,C -1.4832,E1 25.1406,E2 478.2491} C_DIS
LIN {X 107.4036,Y -61.7228,Z 131,A -33.7612,B 24.9588,C -1.4832,E1 25.1381,E2 480.0583} C_DIS
LIN {X 105.6018,Y -64.7573,Z 131,A -35.3281,B 24.9588,C -1.4818,E1 25.1359,E2 481.6206} C_DIS
LIN {X 103.7375,Y -67.7049,Z 131,A -37.11,B 24.9596,C -1.4686,E1 25.1332,E2 483.4248} C_DIS
LIN {X 101.6719,Y -70.768,Z 131,A -38.777,B 24.9597,C -1.4659,E1 25.1305,E2 485.09} C_DIS
LIN {X 99.7379,Y -73.4693,Z 131,A -40.3149,B 24.96,C -1.4615,E1 25.128,E2 486.6307} C_DIS
LIN {X 97.2012,Y -76.7931,Z 131,A -42.1389,B 24.96,C -1.4618,E1 25.1249,E2 488.4455} C_DIS
LIN {X 94.8684,Y -79.6581,Z 131,A -43.7723,B 24.96,C -1.461,E1 25.122,E2 490.0731} C_DIS
LIN {X 92.6982,Y -82.1734,Z 131,A -45.4855,B 24.9607,C -1.4481,E1 25.1188,E2 491.8092} C_DIS
LIN {X 90.2059,Y -84.9008,Z 131,A -47.1534,B 24.9608,C -1.4458,E1 25.1157,E2 493.4751} C_DIS
LIN {X 87.2896,Y -87.8971,Z 131,A -49.0923,B 24.9611,C -1.4407,E1 25.1119,E2 495.4178} C_DIS
LIN {X 84.6295,Y -90.4611,Z 131,A -50.7875,B 24.9613,C -1.4373,E1 25.1084,E2 497.1141} C_DIS
LIN {X 81.5281,Y -93.2654,Z 131,A -52.6102,B 24.9613,C -1.4383,E1 25.1046,E2 498.9271} C_DIS
LIN {X 78.9974,Y -95.4176,Z 131,A -54.1136,B 24.9613,C -1.4365,E1 25.1014,E2 500.4291} C_DIS
LIN {X 76.1175,Y -97.732,Z 131,A -55.9623,B 24.9619,C -1.4257,E1 25.0973,E2 502.2964} C_DIS
LIN {X 73.1688,Y -99.9579,Z 131,A -57.5868,B 24.9619,C -1.4262,E1 25.0937,E2 503.9138} C_DIS
LIN {X 70.4622,Y -101.8844,Z 131,A -59.172,B 24.9622,C -1.4206,E1 25.0901,E2 505.5067} C_DIS
LIN {X 66.9834,Y -104.2041,Z 131,A -61.0083,B 24.9622,C -1.4216,E1 25.0858,E2 507.3346} C_DIS
LIN {X 64.1647,Y -105.9624,Z 131,A -62.5048,B 24.9622,C -1.4207,E1 25.0823,E2 508.8286} C_DIS
LIN {X 60.9768,Y -107.8297,Z 131,A -64.3508,B 24.9627,C -1.4107,E1 25.0777,E2 510.6926} C_DIS
LIN {X 57.7337,Y -109.5995,Z 131,A -65.974,B 24.9627,C -1.412,E1 25.0738,E2 512.3082} C_DIS
LIN {X 54.7741,Y -111.1087,Z 131,A -67.5631,B 24.9629,C -1.4068,E1 25.0698,E2 513.9052} C_DIS
LIN {X 50.993,Y -112.8938,Z 131,A -69.4056,B 24.9629,C -1.4082,E1 25.0651,E2 515.7396} C_DIS
LIN {X 47.6039,Y -114.3647,Z 131,A -71.2043,B 24.9632,C -1.4012,E1 25.0605,E2 517.5505} C_DIS
LIN {X 44.1411,Y -115.744,Z 131,A -72.8904,B 24.9632,C -1.4007,E1 25.0561,E2 519.2343} C_DIS
LIN {X 40.2412,Y -117.1583,Z 131,A -74.8467,B 24.9635,C -1.3963,E1 25.0509,E2 521.1969} C_DIS
LIN {X 36.7293,Y -118.3054,Z 131,A -76.5193,B 24.9635,C -1.396,E1 25.0465,E2 522.8672} C_DIS
LIN {X 32.7159,Y -119.4783,Z 131,A -78.4906,B 24.9637,C -1.392,E1 25.0412,E2 524.8447} C_DIS
LIN {X 29.1383,Y -120.4006,Z 131,A -80.1641,B 24.9637,C -1.392,E1 25.0366,E2 526.5157} C_DIS
LIN {X 25.1123,Y -121.3039,Z 131,A -81.9963,B 24.9637,C -1.394,E1 25.0317,E2 528.3408} C_DIS
LIN {X 21.4294,Y -122.009,Z 131,A -83.8103,B 24.9639,C -1.3887,E1 25.0267,E2 530.1654} C_DIS
LIN {X 17.2995,Y -122.6617,Z 131,A -85.619,B 24.9636,C -1.3934,E1 25.0217,E2 531.9613} C_DIS
LIN {X 13.6339,Y -123.1241,Z 131,A -87.4582,B 24.964,C -1.386,E1 25.0165,E2 533.8166} C_DIS
LIN {X 9.9561,Y -123.475,Z 131,A -89.1333,B 24.964,C -1.3867,E1 25.0119,E2 535.489} C_DIS
LIN {X 5.7833,Y -123.7415,Z 131,A -91.1077,B 24.9641,C -1.384,E1 25.0064,E2 537.4692} C_DIS
LIN {X 2.0906,Y -123.8586,Z 131,A -92.7836,B 24.9641,C -1.385,E1 25.0017,E2 539.1423} C_DIS
LIN {X 2.0906,Y -123.8586,Z 131,A -92.7836,B 24.9641,C -1.385,E1 25.0017,E2 539.1423} C_DIS
Enddeposition()
LIN {X 0.8792,Y -123.0306,Z 131,A -93.2479,B 24.9631,C -1.4043,E1 25.0005,E2 539.5607} C_DIS
Startdeposition()
$VEL.CP = VEL_PRINT
LIN {X 5.6184,Y -122.9071,Z 131,A -90.3621,B 24.9613,C -1.4375,E1 25.0088,E2 536.5969} C_DIS
LIN {X 9.3066,Y -122.6826,Z 131,A -88.6865,B 24.9613,C -1.4361,E1 25.0135,E2 534.9253} C_DIS
LIN {X 12.8162,Y -122.3655,Z 131,A -87.1067,B 24.9615,C -1.4341,E1 25.0178,E2 533.3515} C_DIS
LIN {X 15.8776,Y -122.0064,Z 131,A -85.1749,B 24.9601,C -1.4592,E1 25.0234,E2 531.3617} C_DIS
LIN {X 19.546,Y -121.4726,Z 131,A -83.8133,B 24.961,C -1.4426,E1 25.027,E2 530.0407} C_DIS
LIN {X 23.3772,Y -120.7939,Z 131,A -81.9755,B 24.9609,C -1.4454,E1 25.0321,E2 528.1984} C_DIS
LIN {X 26.1286,Y -120.2284,Z 131,A -80.3498,B 24.9599,C -1.4622,E1 25.0366,E2 526.535} C_DIS
LIN {X 29.6941,Y -119.3979,Z 131,A -78.9585,B 24.9607,C -1.4485,E1 25.0403,E2 525.1783} C_DIS
LIN {X 33.6108,Y -118.3556,Z 131,A -77.0913,B 24.9607,C -1.4495,E1 25.0453,E2 523.3116} C_DIS
LIN {X 36.3729,Y -117.5356,Z 131,A -75.6892,B 24.9604,C -1.4541,E1 25.0491,E2 521.9011} C_DIS
LIN {X 40.7295,Y -116.098,Z 131,A -73.6829,B 24.9606,C -1.4504,E1 25.0543,E2 519.9076} C_DIS
LIN {X 44.3688,Y -114.7568,Z 131,A -71.8403,B 24.9604,C -1.4547,E1 25.0592,E2 518.0588} C_DIS
LIN {X 51.3382,Y -111.813,Z 131,A -68.1285,B 24.9596,C -1.4693,E1 25.0687,E2 514.3212} C_DIS
LIN {X 55.9033,Y -109.6009,Z 131,A -66.006,B 24.96,C -1.4613,E1 25.074,E2 512.2234} C_DIS
LIN {X 59.3975,Y -107.7483,Z 131,A -63.6341,B 24.9583,C -1.4911,E1 25.0799,E2 509.788} C_DIS
LIN {X 63.2161,Y -105.5528,Z 131,A -62.0787,B 24.9595,C -1.4701,E1 25.0836,E2 508.2872} C_DIS
LIN {X 66.5712,Y -103.4696,Z 131,A -60.2946,B 24.9595,C -1.4709,E1 25.0877,E2 506.5068} C_DIS
LIN {X 70.3028,Y -100.9713,Z 131,A -58.1917,B 24.9592,C -1.4757,E1 25.0926,E2 504.3996} C_DIS
LIN {X 73.4703,Y -98.6902,Z 131,A -56.389,B 24.959,C -1.4788,E1 25.0967,E2 502.596} C_DIS
LIN {X 76.1634,Y -96.6269,Z 131,A -54.8484,B 24.959,C -1.4803,E1 25.1001,E2 501.0575} C_DIS
LIN {X 79.2396,Y -94.1212,Z 131,A -52.9925,B 24.9587,C -1.4849,E1 25.1041,E2 499.1979} C_DIS
LIN {X 82.096,Y -91.6391,Z 131,A -51.2356,B 24.9585,C -1.4888,E1 25.1077,E2 497.4388} C_DIS
LIN {X 84.9524,Y -88.9996,Z 131,A -49.3381,B 24.958,C -1.4975,E1 25.1116,E2 495.5285} C_DIS
LIN {X 87.9147,Y -86.0734,Z 131,A -47.6652,B 24.9585,C -1.4889,E1 25.1149,E2 493.883} C_DIS
LIN {X 89.5981,Y -84.3197,Z 131,A -46.2833,B 24.9576,C -1.5044,E1 25.1176,E2 492.4706} C_DIS
LIN {X 92.4623,Y -81.1684,Z 131,A -44.4296,B 24.9576,C -1.503,E1 25.121,E2 490.6284} C_DIS
LIN {X 94.9936,Y -78.1923,Z 131,A -42.557,B 24.9573,C -1.5105,E1 25.1244,E2 488.7467} C_DIS
LIN {X 97.6783,Y -74.8102,Z 131,A -40.2891,B 24.9562,C -1.5291,E1 25.1283,E2 486.4456} C_DIS
LIN {X 99.6942,Y -72.1026,Z 131,A -38.4473,B 24.9551,C -1.5474,E1 25.1314,E2 484.5697} C_DIS
LIN {X 102.3806,Y -68.2351,Z 131,A -37.003,B 24.957,C -1.5153,E1 25.1335,E2 483.2082} C_DIS
LIN {X 105.4527,Y -63.3841,Z 131,A -34.1142,B 24.9559,C -1.534,E1 25.1378,E2 480.29} C_DIS
LIN {X 107.7129,Y -59.4621,Z 131,A -32.0505,B 24.9557,C -1.538,E1 25.1407,E2 478.2277} C_DIS
LIN {X 109.3623,Y -56.3694,Z 131,A -30.0754,B 24.9544,C -1.5605,E1 25.1432,E2 476.2099} C_DIS
LIN {X 111.0489,Y -52.9689,Z 131,A -28.8464,B 24.9557,C -1.5382,E1 25.1447,E2 475.0399} C_DIS
LIN {X 112.6977,Y -49.3652,Z 131,A -26.8358,B 24.9548,C -1.5524,E1 25.147,E2 473.0069} C_DIS
LIN {X 114.3059,Y -45.5175,Z 131,A -24.9026,B 24.9545,C -1.558,E1 25.149,E2 471.0712} C_DIS
LIN {X 115.3269,Y -42.8647,Z 131,A -23.4408,B 24.9539,C -1.5692,E1 25.1505,E2 469.5911} C_DIS
LIN {X 116.9302,Y -38.2746,Z 131,A -21.3638,B 24.954,C -1.5668,E1 25.1523,E2 467.5315} C_DIS
LIN {X 117.8931,Y -35.1957,Z 131,A -19.4666,B 24.9525,C -1.5919,E1 25.1539,E2 465.5859} C_DIS
LIN {X 118.9806,Y -31.3264,Z 131,A -17.4504,B 24.9517,C -1.6054,E1 25.1553,E2 463.5494} C_DIS
LIN {X 120.0948,Y -26.738,Z 131,A -15.8199,B 24.953,C -1.5833,E1 25.1563,E2 461.9807} C_DIS
LIN {X 120.7127,Y -23.7939,Z 131,A -14.43,B 24.9528,C -1.5873,E1 25.157,E2 460.5895} C_DIS
LIN {X 121.3584,Y -20.245,Z 131,A -12.7866,B 24.9526,C -1.5909,E1 25.1578,E2 458.9472} C_DIS
LIN {X 121.953,Y -16.2808,Z 131,A -10.9112,B 24.9522,C -1.5975,E1 25.1586,E2 457.0673} C_DIS
LIN {X 122.4307,Y -12.1835,Z 131,A -9.2433,B 24.9526,C -1.5908,E1 25.1591,E2 455.425} C_DIS
LIN {X 122.69,Y -9.2123,Z 131,A -7.6014,B 24.9515,C -1.6083,E1 25.1594,E2 453.7515} C_DIS
LIN {X 122.8797,Y -6.1807,Z 131,A -6.1964,B 24.9513,C -1.6125,E1 25.1597,E2 452.3451} C_DIS
LIN {X 123.0198,Y -1.9525,Z 131,A -4.3207,B 24.9512,C -1.6141,E1 25.1597,E2 450.4767} C_DIS
LIN {X 123.0292,Y 1.2713,Z 131,A -2.8303,B 24.9509,C -1.6185,E1 25.1597,E2 448.9849} C_DIS
LIN {X 122.9432,Y 4.7551,Z 131,A -1.2519,B 24.9507,C -1.6215,E1 25.1597,E2 447.4088} C_DIS
LIN {X 122.7654,Y 8.141,Z 131,A 0.4037,B 24.9502,C -1.6306,E1 25.1593,E2 445.7416} C_DIS
LIN {X 122.4239,Y 12.2542,Z 131,A 2.415,B 24.9495,C -1.6414,E1 25.1588,E2 443.7168} C_DIS
LIN {X 121.7783,Y 17.5382,Z 131,A 4.7752,B 24.9494,C -1.6433,E1 25.158,E2 441.3659} C_DIS
LIN {X 121.1255,Y 21.5923,Z 131,A 6.6925,B 24.949,C -1.6496,E1 25.1571,E2 439.4449} C_DIS
LIN {X 120.1952,Y 26.2796,Z 131,A 9.0977,B 24.948,C -1.6659,E1 25.1557,E2 437.0154} C_DIS
LIN {X 119.0399,Y 31.0991,Z 131,A 11.2128,B 24.9482,C -1.6632,E1 25.1542,E2 434.9188} C_DIS
LIN {X 117.9037,Y 35.1603,Z 131,A 13.1061,B 24.948,C -1.6657,E1 25.1528,E2 433.0305} C_DIS
LIN {X 116.6652,Y 39.075,Z 131,A 15.0265,B 24.9476,C -1.672,E1 25.1511,E2 431.1062} C_DIS
LIN {X 115.2567,Y 43.0547,Z 131,A 17.2404,B 24.9464,C -1.6905,E1 25.149,E2 428.861} C_DIS
LIN {X 114.0869,Y 46.0639,Z 131,A 18.4888,B 24.947,C -1.682,E1 25.1477,E2 427.6396} C_DIS
LIN {X 112.5,Y 49.8134,Z 131,A 20.2809,B 24.947,C -1.6822,E1 25.1457,E2 425.8566} C_DIS
LIN {X 111.0019,Y 53.0674,Z 131,A 22.064,B 24.9463,C -1.6929,E1 25.1436,E2 424.0581} C_DIS
LIN {X 109.1027,Y 56.8702,Z 131,A 23.9734,B 24.9462,C -1.6949,E1 25.1412,E2 422.1541} C_DIS
LIN {X 107.3154,Y 60.1741,Z 131,A 25.8184,B 24.9455,C -1.7046,E1 25.1386,E2 420.2958} C_DIS
LIN {X 105.028,Y 64.0831,Z 131,A 27.8239,B 24.9455,C -1.7051,E1 25.1358,E2 418.2995} C_DIS
LIN {X 103.0048,Y 67.289,Z 131,A 29.4292,B 24.9457,C -1.7017,E1 25.1334,E2 416.7103} C_DIS
LIN {X 101.1783,Y 70.0052,Z 131,A 31.1129,B 24.945,C -1.7136,E1 25.1307,E2 415.0066} C_DIS
LIN {X 98.8865,Y 73.2059,Z 131,A 32.9461,B 24.9447,C -1.7183,E1 25.1277,E2 413.1713} C_DIS
LIN {X 96.5004,Y 76.324,Z 131,A 34.7633,B 24.9444,C -1.7222,E1 25.1246,E2 411.3535} C_DIS
LIN {X 93.7733,Y 79.6503,Z 131,A 36.7056,B 24.9444,C -1.7239,E1 25.1211,E2 409.4159} C_DIS
LIN {X 91.1381,Y 82.6532,Z 131,A 38.5838,B 24.944,C -1.7291,E1 25.1176,E2 407.534} C_DIS
LIN {X 88.359,Y 85.617,Z 131,A 40.3872,B 24.944,C -1.7289,E1 25.1141,E2 405.7388} C_DIS
LIN {X 85.9592,Y 88.0268,Z 131,A 42.0489,B 24.9435,C -1.7362,E1 25.1108,E2 404.067} C_DIS
LIN {X 83.2579,Y 90.5859,Z 131,A 43.7291,B 24.9435,C -1.7372,E1 25.1074,E2 402.3912} C_DIS
LIN {X 80.4977,Y 93.0471,Z 131,A 45.5104,B 24.943,C -1.7436,E1 25.1036,E2 400.6018} C_DIS
LIN {X 77.3573,Y 95.6743,Z 131,A 47.3806,B 24.943,C -1.7454,E1 25.0996,E2 398.7344} C_DIS
LIN {X 74.2432,Y 98.1098,Z 131,A 49.2351,B 24.9426,C -1.7495,E1 25.0955,E2 396.8771} C_DIS
LIN {X 70.8999,Y 100.5533,Z 131,A 50.8822,B 24.9433,C -1.739,E1 25.0918,E2 395.2606} C_DIS
LIN {X 68.4724,Y 102.2213,Z 131,A 52.5259,B 24.9423,C -1.7547,E1 25.088,E2 393.5854} C_DIS
LIN {X 64.9632,Y 104.4862,Z 131,A 54.1536,B 24.9431,C -1.7422,E1 25.0842,E2 391.9923} C_DIS
LIN {X 62.5433,Y 105.9531,Z 131,A 55.7664,B 24.942,C -1.7586,E1 25.0803,E2 390.3458} C_DIS
LIN {X 59.0038,Y 107.9637,Z 131,A 57.645,B 24.942,C -1.7605,E1 25.0757,E2 388.4683} C_DIS
LIN {X 55.4649,Y 109.8247,Z 131,A 59.3032,B 24.9424,C -1.753,E1 25.0716,E2 386.8324} C_DIS
LIN {X 52.6897,Y 111.1822,Z 131,A 60.9676,B 24.9416,C -1.7658,E1 25.0674,E2 385.1422} C_DIS
LIN {X 49.3144,Y 112.7199,Z 131,A 62.4523,B 24.9422,C -1.756,E1 25.0637,E2 383.6842} C_DIS
LIN {X 46.0568,Y 114.0898,Z 131,A 64.3321,B 24.9413,C -1.7691,E1 25.0587,E2 381.7778} C_DIS
LIN {X 42.352,Y 115.5162,Z 131,A 66.1512,B 24.9413,C -1.7694,E1 25.054,E2 379.9617} C_DIS
LIN {X 38.7886,Y 116.7616,Z 131,A 67.9302,B 24.9412,C -1.772,E1 25.0493,E2 378.1803} C_DIS
LIN {X 34.4419,Y 118.1167,Z 131,A 70.0074,B 24.9412,C -1.7715,E1 25.0437,E2 376.1079} C_DIS
LIN {X 31.5348,Y 118.9253,Z 131,A 71.7017,B 24.9402,C -1.7863,E1 25.0391,E2 374.3811} C_DIS
LIN {X 28.2603,Y 119.7458,Z 131,A 72.8596,B 24.9415,C -1.7674,E1 25.0361,E2 373.2699} C_DIS
LIN {X 24.1982,Y 120.6319,Z 131,A 74.9133,B 24.941,C -1.7739,E1 25.0304,E2 371.2032} C_DIS
LIN {X 20.6043,Y 121.2976,Z 131,A 76.6761,B 24.9408,C -1.7774,E1 25.0255,E2 369.434} C_DIS
LIN {X 16.4771,Y 121.9267,Z 131,A 78.5249,B 24.9411,C -1.7734,E1 25.0205,E2 367.5963} C_DIS
LIN {X 12.8531,Y 122.3615,Z 131,A 80.272,B 24.9409,C -1.776,E1 25.0156,E2 365.8444} C_DIS
LIN {X 9.1019,Y 122.6986,Z 131,A 81.8293,B 24.9415,C -1.7668,E1 25.0113,E2 364.3097} C_DIS
LIN {X 6.4593,Y 122.8656,Z 131,A 83.2827,B 24.9408,C -1.7772,E1 25.0072,E2 362.8322} C_DIS
LIN {X 2.2205,Y 123.0154,Z 131,A 85.1914,B 24.941,C -1.7738,E1 25.0019,E2 360.9318} C_DIS
LIN {X -1.7406,Y 123.0227,Z 131,A 87.0406,B 24.941,C -1.7736,E1 24.9967,E2 359.0831} C_DIS
LIN {X -6.0847,Y 122.8845,Z 131,A 89.0128,B 24.9412,C -1.7706,E1 24.9913,E2 357.1178} C_DIS
LIN {X -9.1777,Y 122.6927,Z 131,A 90.6076,B 24.9408,C -1.777,E1 24.9868,E2 355.507} C_DIS
LIN {X -13.1334,Y 122.3318,Z 131,A 92.4178,B 24.941,C -1.7742,E1 24.9818,E2 353.7025} C_DIS
LIN {X -17.2214,Y 121.8237,Z 131,A 94.2457,B 24.9414,C -1.7688,E1 24.9767,E2 351.8861} C_DIS
LIN {X -21.1167,Y 121.2097,Z 131,A 96.123,B 24.9414,C -1.7694,E1 24.9716,E2 350.0057} C_DIS
LIN {X -26.3433,Y 120.1813,Z 131,A 98.6324,B 24.9414,C -1.7686,E1 24.9647,E2 347.4952} C_DIS
LIN {X -30.2457,Y 119.2599,Z 131,A 100.534,B 24.9414,C -1.7684,E1 24.9595,E2 345.5915} C_DIS
LIN {X -34.2925,Y 118.1597,Z 131,A 102.4668,B 24.9416,C -1.7653,E1 24.9543,E2 343.6628} C_DIS
LIN {X -38.1081,Y 116.9848,Z 131,A 104.8198,B 24.9402,C -1.7859,E1 24.9479,E2 341.2566} C_DIS
LIN {X -42.2018,Y 115.5713,Z 131,A 106.1002,B 24.9426,C -1.7494,E1 24.9448,E2 340.0604} C_DIS
LIN {X -47.472,Y 113.508,Z 131,A 108.7493,B 24.9428,C -1.7463,E1 24.938,E2 337.4129} C_DIS
LIN {X -51.0973,Y 111.9227,Z 131,A 110.8394,B 24.9423,C -1.7548,E1 24.9325,E2 335.2976} C_DIS
LIN {X -54.4303,Y 110.3409,Z 131,A 112.6015,B 24.9423,C -1.7541,E1 24.9281,E2 333.5327} C_DIS
LIN {X -57.7651,Y 108.6321,Z 131,A 114.2722,B 24.9428,C -1.7477,E1 24.924,E2 331.8725} C_DIS
LIN {X -61.6232,Y 106.4913,Z 131,A 116.3753,B 24.9428,C -1.7463,E1 24.9189,E2 329.7667} C_DIS
LIN {X -64.8201,Y 104.5751,Z 131,A 117.9932,B 24.9434,C -1.7377,E1 24.915,E2 328.1642} C_DIS
LIN {X -67.6829,Y 102.745,Z 131,A 119.688,B 24.9433,C -1.7397,E1 24.911,E2 326.4591} C_DIS
LIN {X -71.0836,Y 100.4233,Z 131,A 121.4278,B 24.9441,C -1.7278,E1 24.9071,E2 324.7418} C_DIS
LIN {X -75.0871,Y 97.4649,Z 131,A 124.4485,B 24.9423,C -1.7546,E1 24.9002,E2 321.6465} C_DIS
LIN {X -78.4309,Y 94.7953,Z 131,A 125.8244,B 24.9444,C -1.7223,E1 24.8974,E2 320.3422} C_DIS
LIN {X -83.6341,Y 90.2385,Z 131,A 129.3563,B 24.944,C -1.7287,E1 24.89,E2 316.781} C_DIS
LIN {X -88.144,Y 85.8398,Z 131,A 132.4106,B 24.9441,C -1.7269,E1 24.8839,E2 313.7181} C_DIS
LIN {X -92.0596,Y 81.6264,Z 131,A 135.4689,B 24.9435,C -1.7371,E1 24.8781,E2 310.6219} C_DIS
LIN {X -95.2176,Y 77.9181,Z 131,A 137.167,B 24.9455,C -1.7055,E1 24.8752,E2 308.9911} C_DIS
LIN {X -97.787,Y 74.6692,Z 131,A 139.0666,B 24.9459,C -1.699,E1 24.872,E2 307.098} C_DIS
LIN {X -100.2172,Y 71.3724,Z 131,A 141.0145,B 24.9461,C -1.6955,E1 24.8688,E2 305.149} C_DIS
LIN {X -102.6285,Y 67.8594,Z 131,A 142.9088,B 24.9467,C -1.686,E1 24.8659,E2 303.268} C_DIS
LIN {X -106.4973,Y 61.6126,Z 131,A 146.5503,B 24.9467,C -1.6857,E1 24.8606,E2 299.6084} C_DIS
LIN {X -108.627,Y 57.7745,Z 131,A 148.55,B 24.9473,C -1.6776,E1 24.8579,E2 297.6174} C_DIS
LIN {X -110.59,Y 53.9211,Z 131,A 150.4072,B 24.9481,C -1.6647,E1 24.8556,E2 295.7811} C_DIS
LIN {X -112.0694,Y 50.7749,Z 131,A 151.9888,B 24.9485,C -1.6581,E1 24.8538,E2 294.2066} C_DIS
LIN {X -113.6343,Y 47.1697,Z 131,A 154.0253,B 24.9483,C -1.6615,E1 24.8515,E2 292.1506} C_DIS
LIN {X -115.2097,Y 43.1794,Z 131,A 155.9701,B 24.9488,C -1.6529,E1 24.8496,E2 290.2155} C_DIS
LIN {X -116.4633,Y 39.6723,Z 131,A 157.6628,B 24.9493,C -1.6456,E1 24.848,E2 288.5305} C_DIS
LIN {X -117.5516,Y 36.3209,Z 131,A 159.3131,B 24.9496,C -1.6408,E1 24.8466,E2 286.8822} C_DIS
LIN {X -118.539,Y 32.9562,Z 131,A 161.0475,B 24.9496,C -1.64,E1 24.8453,E2 285.1396} C_DIS
LIN {X -119.7,Y 28.4522,Z 131,A 163.1895,B 24.9501,C -1.632,E1 24.8439,E2 283.0043} C_DIS
LIN {X -120.5241,Y 24.7318,Z 131,A 165.1455,B 24.95,C -1.6342,E1 24.8427,E2 281.0314} C_DIS
LIN {X -121.5064,Y 19.3374,Z 131,A 167.5804,B 24.9508,C -1.6207,E1 24.8416,E2 278.6144} C_DIS
LIN {X -122.053,Y 15.5164,Z 131,A 169.3491,B 24.9512,C -1.6135,E1 24.8409,E2 276.8521} C_DIS
LIN {X -122.6625,Y 9.5631,Z 131,A 172.0792,B 24.9519,C -1.6019,E1 24.8402,E2 274.1333} C_DIS
LIN {X -122.8807,Y 6.1604,Z 131,A 173.8483,B 24.9518,C -1.6046,E1 24.8399,E2 272.347} C_DIS
LIN {X -123.0198,Y 1.948,Z 131,A 175.7109,B 24.9524,C -1.5938,E1 24.8398,E2 270.4991} C_DIS
LIN {X -122.984,Y -3.5496,Z 131,A 178.2918,B 24.9529,C -1.5863,E1 24.8399,E2 267.9205} C_DIS
LIN {X -122.6848,Y -9.2777,Z 131,A -178.9497,B 24.9531,C -1.5814,E1 24.8404,E2 265.1569} C_DIS
LIN {X -122.2865,Y -13.5591,Z 131,A -176.9261,B 24.9535,C -1.5759,E1 24.8409,E2 263.1345} C_DIS
LIN {X -121.7603,Y -17.6633,Z 131,A -175.0027,B 24.9538,C -1.5696,E1 24.8417,E2 261.2147} C_DIS
LIN {X -121.1025,Y -21.7199,Z 131,A -173.1664,B 24.9544,C -1.56,E1 24.8425,E2 259.3902} C_DIS
LIN {X -120.3962,Y -25.3448,Z 131,A -171.3209,B 24.9544,C -1.5601,E1 24.8435,E2 257.5336} C_DIS
LIN {X -119.5276,Y -29.1696,Z 131,A -169.4661,B 24.9547,C -1.5557,E1 24.8447,E2 255.6785} C_DIS
LIN {X -118.3676,Y -33.5684,Z 131,A -167.3332,B 24.955,C -1.5497,E1 24.8463,E2 253.5474} C_DIS
LIN {X -117.0758,Y -37.8284,Z 131,A -165.279,B 24.9554,C -1.5426,E1 24.848,E2 251.4985} C_DIS
LIN {X -115.6836,Y -41.8923,Z 131,A -163.2447,B 24.9557,C -1.538,E1 24.8499,E2 249.4634} C_DIS
LIN {X -114.1772,Y -45.8386,Z 131,A -161.1894,B 24.9557,C -1.5361,E1 24.852,E2 247.4012} C_DIS
LIN {X -112.3914,Y -50.058,Z 131,A -159.234,B 24.9566,C -1.522,E1 24.8541,E2 245.4687} C_DIS
LIN {X -110.9711,Y -53.1318,Z 131,A -157.5392,B 24.9566,C -1.5227,E1 24.8562,E2 243.7629} C_DIS
LIN {X -108.9637,Y -57.1357,Z 131,A -154.5373,B 24.9545,C -1.5582,E1 24.8602,E2 240.6605} C_DIS
LIN {X -105.8621,Y -62.6964,Z 131,A -152.4387,B 24.9572,C -1.5109,E1 24.863,E2 238.6636} C_DIS
LIN {X -103.5914,Y -66.3817,Z 131,A -150.4315,B 24.9576,C -1.5051,E1 24.866,E2 236.66} C_DIS
LIN {X -101.3719,Y -69.7235,Z 131,A -148.5597,B 24.9578,C -1.5005,E1 24.8689,E2 234.7899} C_DIS
LIN {X -99.2567,Y -72.7034,Z 131,A -146.8489,B 24.958,C -1.4966,E1 24.8717,E2 233.0801} C_DIS
LIN {X -96.9472,Y -75.7557,Z 131,A -144.981,B 24.958,C -1.4961,E1 24.8749,E2 231.2046} C_DIS
LIN {X -94.1283,Y -79.2312,Z 131,A -142.9752,B 24.9585,C -1.4876,E1 24.8784,E2 229.2096} C_DIS
LIN {X -91.5931,Y -82.1475,Z 131,A -141.1337,B 24.9587,C -1.4853,E1 24.8819,E2 227.3652} C_DIS
LIN {X -88.7066,Y -85.2564,Z 131,A -139.1644,B 24.9589,C -1.4807,E1 24.8856,E2 225.3985} C_DIS
LIN {X -85.7298,Y -88.2502,Z 131,A -137.0663,B 24.9589,C -1.4825,E1 24.8898,E2 223.2873} C_DIS
LIN {X -82.2827,Y -91.472,Z 131,A -135.0289,B 24.9595,C -1.4707,E1 24.894,E2 221.2697} C_DIS
LIN {X -79.2617,Y -94.1025,Z 131,A -133.0809,B 24.9595,C -1.4707,E1 24.8981,E2 219.3139} C_DIS
LIN {X -76.0033,Y -96.7527,Z 131,A -131.2313,B 24.9599,C -1.4623,E1 24.9021,E2 217.4776} C_DIS
LIN {X -73.3075,Y -98.8111,Z 131,A -129.2022,B 24.959,C -1.4802,E1 24.9068,E2 215.3987} C_DIS
LIN {X -70.2423,Y -101.0135,Z 131,A -127.7735,B 24.96,C -1.462,E1 24.91,E2 214.0084} C_DIS
LIN {X -67.6241,Y -102.7838,Z 131,A -126.1853,B 24.9598,C -1.465,E1 24.9137,E2 212.4079} C_DIS
LIN {X -63.8569,Y -105.1656,Z 131,A -124.2267,B 24.9603,C -1.4564,E1 24.9183,E2 210.4635} C_DIS
LIN {X -60.2575,Y -107.2688,Z 131,A -122.3143,B 24.9605,C -1.4523,E1 24.9229,E2 208.5553} C_DIS
LIN {X -57.4947,Y -108.7753,Z 131,A -120.7336,B 24.9603,C -1.4556,E1 24.9269,E2 206.9621} C_DIS
LIN {X -53.5587,Y -110.7665,Z 131,A -118.768,B 24.9607,C -1.449,E1 24.9318,E2 205.0072} C_DIS
LIN {X -49.6651,Y -112.5659,Z 131,A -116.8133,B 24.9609,C -1.4447,E1 24.9367,E2 203.0579} C_DIS
LIN {X -46.5729,Y -113.8799,Z 131,A -115.2132,B 24.9609,C -1.4447,E1 24.9409,E2 201.4541} C_DIS
LIN {X -42.8911,Y -115.3172,Z 131,A -113.3291,B 24.9609,C -1.445,E1 24.9458,E2 199.5654} C_DIS
LIN {X -39.0618,Y -116.6697,Z 131,A -111.4483,B 24.9609,C -1.4429,E1 24.9507,E2 197.6859} C_DIS
LIN {X -35.0318,Y -117.9419,Z 131,A -109.789,B 24.9619,C -1.4269,E1 24.9551,E2 196.0616} C_DIS
LIN {X -31.0287,Y -119.0581,Z 131,A -107.7953,B 24.9618,C -1.4284,E1 24.9605,E2 194.0614} C_DIS
LIN {X -27.9286,Y -119.8236,Z 131,A -106.0417,B 24.9611,C -1.4402,E1 24.9653,E2 192.2774} C_DIS
LIN {X -23.6887,Y -120.7339,Z 131,A -103.9544,B 24.9611,C -1.4425,E1 24.971,E2 190.1822} C_DIS
LIN {X -19.2978,Y -121.5128,Z 131,A -101.9474,B 24.9612,C -1.4386,E1 24.9765,E2 188.1827} C_DIS
LIN {X -15.7676,Y -122.0209,Z 131,A -100.3111,B 24.9613,C -1.437,E1 24.9811,E2 186.5487} C_DIS
LIN {X -12.3351,Y -122.416,Z 131,A -98.7507,B 24.9615,C -1.4345,E1 24.9854,E2 184.9933} C_DIS
LIN {X -9.3759,Y -122.6772,Z 131,A -97.4273,B 24.9616,C -1.4316,E1 24.9891,E2 183.6763} C_DIS
LIN {X -6.1357,Y -122.8819,Z 131,A -95.8083,B 24.9613,C -1.4368,E1 24.9936,E2 182.0444} C_DIS
LIN {X -2.5952,Y -123.0078,Z 131,A -94.1605,B 24.9613,C -1.4369,E1 24.9982,E2 180.3961} C_DIS
LIN {X 0.8792,Y -123.0306,Z 131,A -93.2461,B 24.9631,C -1.4036,E1 25.0005,E2 179.5607} C_DIS
Enddeposition()
LIN {X 0.8792,Y -123.0306,Z 131,A -93.2461,B 24.9631,C -1.4036,E1 25.0005,E2 179.5607} C_DIS
Startdeposition()
$VEL.CP = VEL_PRINT
LIN {X -1.8654,Y -122.1803,Z 131,A -94.6454,B 24.9626,C -1.4129,E1 24.9967,E2 180.9382} C_DIS
LIN {X -5.5731,Y -122.0677,Z 131,A -96.6163,B 24.9632,C -1.4018,E1 24.9911,E2 182.9356} C_DIS
LIN {X -11.1983,Y -121.6806,Z 131,A -98.7838,B 24.962,C -1.4242,E1 24.9852,E2 185.051} C_DIS
LIN {X -15.7051,Y -121.1814,Z 131,A -101.2055,B 24.9627,C -1.4107,E1 24.9784,E2 187.5063} C_DIS
LIN {X -20.0263,Y -120.5425,Z 131,A -103.6141,B 24.9636,C -1.3946,E1 24.9717,E2 189.9552} C_DIS
LIN {X -23.7158,Y -119.8712,Z 131,A -104.9397,B 24.9625,C -1.4152,E1 24.9682,E2 191.2332} C_DIS
LIN {X -29.2605,Y -118.6394,Z 131,A -107.3308,B 24.9617,C -1.4292,E1 24.9617,E2 193.5944} C_DIS
LIN {X -34.1927,Y -117.3136,Z 131,A -110.1066,B 24.9626,C -1.4131,E1 24.9541,E2 196.4126} C_DIS
LIN {X -38.1527,Y -116.0854,Z 131,A -112.0474,B 24.9626,C -1.4148,E1 24.949,E2 198.353} C_DIS
LIN {X -42.1456,Y -114.6963,Z 131,A -114.0161,B 24.9624,C -1.4171,E1 24.9438,E2 200.3199} C_DIS
LIN {X -46.0628,Y -113.1803,Z 131,A -115.9974,B 24.9624,C -1.4186,E1 24.9387,E2 202.3022} C_DIS
LIN {X -51.8231,Y -110.6606,Z 131,A -118.6965,B 24.9615,C -1.4332,E1 24.9319,E2 204.9729} C_DIS
LIN {X -56.9262,Y -108.1245,Z 131,A -121.2506,B 24.9611,C -1.4419,E1 24.9255,E2 207.5131} C_DIS
LIN {X -60.9256,Y -105.9226,Z 131,A -123.7437,B 24.9618,C -1.4289,E1 24.9193,E2 210.0444} C_DIS
LIN {X -64.2533,Y -103.9375,Z 131,A -125.8611,B 24.9623,C -1.4181,E1 24.9142,E2 212.194} C_DIS
LIN {X -67.0457,Y -102.1583,Z 131,A -126.8423,B 24.9608,C -1.4463,E1 24.9121,E2 213.1113} C_DIS
LIN {X -73.1457,Y -97.8843,Z 131,A -130.4311,B 24.9608,C -1.4478,E1 24.9039,E2 216.7088} C_DIS
LIN {X -75.5006,Y -96.0785,Z 131,A -132.0556,B 24.9612,C -1.4399,E1 24.9002,E2 218.3581} C_DIS
LIN {X -78.6654,Y -93.5059,Z 131,A -133.9983,B 24.961,C -1.4422,E1 24.896,E2 220.3027} C_DIS
LIN {X -81.7772,Y -90.7962,Z 131,A -135.9328,B 24.9608,C -1.4461,E1 24.892,E2 222.2356} C_DIS
LIN {X -86.034,Y -86.7741,Z 131,A -138.3839,B 24.9598,C -1.465,E1 24.8871,E2 224.6519} C_DIS
LIN {X -89.2105,Y -83.5051,Z 131,A -140.8611,B 24.9604,C -1.4546,E1 24.8822,E2 227.1645} C_DIS
LIN {X -92.4694,Y -79.8805,Z 131,A -143.0121,B 24.9597,C -1.4658,E1 24.8783,E2 229.2985} C_DIS
LIN {X -94.8753,Y -77.0078,Z 131,A -145.1899,B 24.9605,C -1.4515,E1 24.8744,E2 231.5204} C_DIS
LIN {X -97.0339,Y -74.2693,Z 131,A -146.2881,B 24.959,C -1.4791,E1 24.8726,E2 232.5582} C_DIS
LIN {X -98.7751,Y -71.9369,Z 131,A -147.8811,B 24.9594,C -1.4725,E1 24.8699,E2 234.1747} C_DIS
LIN {X -101.0979,Y -68.6351,Z 131,A -149.7667,B 24.9591,C -1.4776,E1 24.8669,E2 236.0573} C_DIS
LIN {X -103.1971,Y -65.4356,Z 131,A -151.5505,B 24.9588,C -1.4828,E1 24.8642,E2 237.8378} C_DIS
LIN {X -105.2779,Y -62.0335,Z 131,A -153.692,B 24.9592,C -1.476,E1 24.8611,E2 240.0065} C_DIS
LIN {X -108.3279,Y -56.5378,Z 131,A -156.4052,B 24.9582,C -1.4944,E1 24.8575,E2 242.6903} C_DIS
LIN {X -110.0466,Y -53.1159,Z 131,A -158.2585,B 24.958,C -1.4969,E1 24.8552,E2 244.5475} C_DIS
LIN {X -111.7877,Y -49.3462,Z 131,A -160.2365,B 24.9578,C -1.5012,E1 24.853,E2 246.5262} C_DIS
LIN {X -114.0768,Y -43.7955,Z 131,A -162.9022,B 24.9569,C -1.516,E1 24.8502,E2 249.1714} C_DIS
LIN {X -115.2704,Y -40.5492,Z 131,A -164.5187,B 24.9567,C -1.5211,E1 24.8487,E2 250.7849} C_DIS
LIN {X -116.1562,Y -37.9368,Z 131,A -165.9159,B 24.9567,C -1.5205,E1 24.8474,E2 252.1915} C_DIS
LIN {X -117.2684,Y -34.3469,Z 131,A -168.0315,B 24.9572,C -1.5107,E1 24.8457,E2 254.3428} C_DIS
LIN {X -118.168,Y -31.1131,Z 131,A -169.3368,B 24.9563,C -1.5271,E1 24.8448,E2 255.6165} C_DIS
LIN {X -119.1209,Y -27.2326,Z 131,A -171.2348,B 24.956,C -1.532,E1 24.8435,E2 257.5141} C_DIS
LIN {X -119.9851,Y -23.1312,Z 131,A -173.1983,B 24.9557,C -1.5383,E1 24.8425,E2 259.4741} C_DIS
LIN {X -120.7193,Y -18.9314,Z 131,A -175.2272,B 24.9554,C -1.5434,E1 24.8415,E2 261.503} C_DIS
LIN {X -121.2835,Y -14.8941,Z 131,A -177.1548,B 24.9551,C -1.5488,E1 24.8408,E2 263.4291} C_DIS
LIN {X -121.7177,Y -10.7829,Z 131,A -179.1372,B 24.9548,C -1.5532,E1 24.8403,E2 265.4129} C_DIS
LIN {X -122.0396,Y -6.1479,Z 131,A 178.7776,B 24.9542,C -1.5643,E1 24.8399,E2 267.4842} C_DIS
LIN {X -122.1672,Y -2.5858,Z 131,A 177.0254,B 24.954,C -1.5663,E1 24.8399,E2 269.2423} C_DIS
LIN {X -122.1939,Y 0.3106,Z 131,A 175.7115,B 24.9537,C -1.5726,E1 24.8398,E2 270.549} C_DIS
LIN {X -122.1179,Y 4.3323,Z 131,A 173.7654,B 24.9535,C -1.5762,E1 24.8399,E2 272.4983} C_DIS
LIN {X -121.9012,Y 8.4551,Z 131,A 171.7248,B 24.9533,C -1.5781,E1 24.8403,E2 274.5467} C_DIS
LIN {X -121.4932,Y 13.0695,Z 131,A 169.8291,B 24.9522,C -1.597,E1 24.8408,E2 276.4085} C_DIS
LIN {X -121.1185,Y 16.1792,Z 131,A 168.1065,B 24.9526,C -1.5909,E1 24.8414,E2 278.1559} C_DIS
LIN {X -120.4894,Y 20.3435,Z 131,A 166.1573,B 24.9521,C -1.5985,E1 24.8423,E2 280.0988} C_DIS
LIN {X -119.733,Y 24.4053,Z 131,A 164.2125,B 24.9518,C -1.6044,E1 24.8433,E2 282.0409} C_DIS
LIN {X -118.9216,Y 28.0926,Z 131,A 162.0005,B 24.9526,C -1.5913,E1 24.8447,E2 284.297} C_DIS
LIN {X -117.9374,Y 31.9731,Z 131,A 160.6141,B 24.9509,C -1.6183,E1 24.8457,E2 285.6273} C_DIS
LIN {X -116.933,Y 35.4727,Z 131,A 158.8469,B 24.9508,C -1.6212,E1 24.8471,E2 287.3979} C_DIS
LIN {X -115.8264,Y 38.9316,Z 131,A 157.136,B 24.9504,C -1.6262,E1 24.8485,E2 289.1065} C_DIS
LIN {X -114.408,Y 42.9227,Z 131,A 155.3369,B 24.9496,C -1.6405,E1 24.8502,E2 290.8817} C_DIS
LIN {X -113.3231,Y 45.7101,Z 131,A 153.6783,B 24.95,C -1.6339,E1 24.852,E2 292.5654} C_DIS
LIN {X -110.9503,Y 51.2015,Z 131,A 151.0974,B 24.9489,C -1.6521,E1 24.8548,E2 295.1171} C_DIS
LIN {X -109.7177,Y 53.7913,Z 131,A 149.5463,B 24.9492,C -1.6473,E1 24.8567,E2 296.6881} C_DIS
LIN {X -107.9427,Y 57.2715,Z 131,A 147.6156,B 24.9491,C -1.6485,E1 24.8592,E2 298.6261} C_DIS
LIN {X -105.5988,Y 61.4847,Z 131,A 145.3161,B 24.9488,C -1.6535,E1 24.8624,E2 300.9257} C_DIS
LIN {X -102.935,Y 65.8481,Z 131,A 143.1049,B 24.9478,C -1.6685,E1 24.8656,E2 303.1126} C_DIS
LIN {X -100.5533,Y 69.4305,Z 131,A 141.2122,B 24.9471,C -1.6795,E1 24.8686,E2 304.9883} C_DIS
LIN {X -98.9667,Y 71.6736,Z 131,A 139.6927,B 24.9475,C -1.6731,E1 24.8711,E2 306.5306} C_DIS
LIN {X -96.4657,Y 75.0064,Z 131,A 137.864,B 24.9469,C -1.6838,E1 24.8741,E2 308.3425} C_DIS
LIN {X -93.9926,Y 78.0816,Z 131,A 135.454,B 24.9481,C -1.6646,E1 24.8785,E2 310.8095} C_DIS
LIN {X -91.478,Y 81.0149,Z 131,A 133.463,B 24.9483,C -1.6615,E1 24.8822,E2 312.8167} C_DIS
LIN {X -88.3764,Y 84.3875,Z 131,A 132.04,B 24.9459,C -1.6983,E1 24.8848,E2 314.1584} C_DIS
LIN {X -83.0746,Y 89.6108,Z 131,A 127.8086,B 24.9475,C -1.6746,E1 24.8934,E2 318.4639} C_DIS
LIN {X -79.7053,Y 92.6205,Z 131,A 126.3882,B 24.9452,C -1.7098,E1 24.8963,E2 319.8061} C_DIS
LIN {X -76.8371,Y 95.013,Z 131,A 123.5139,B 24.9481,C -1.6649,E1 24.9028,E2 322.7979} C_DIS
LIN {X -71.7298,Y 98.9258,Z 131,A 121.7657,B 24.9441,C -1.7265,E1 24.9064,E2 324.4059} C_DIS
LIN {X -68.664,Y 101.0783,Z 131,A 119.6447,B 24.9449,C -1.714,E1 24.9113,E2 326.5638} C_DIS
LIN {X -63.9199,Y 104.1433,Z 131,A 117.2176,B 24.944,C -1.7288,E1 24.917,E2 328.9634} C_DIS
LIN {X -58.6418,Y 107.2035,Z 131,A 114.2464,B 24.944,C -1.729,E1 24.9242,E2 331.9428} C_DIS
LIN {X -55.3612,Y 108.9339,Z 131,A 112.3516,B 24.9442,C -1.725,E1 24.9289,E2 333.8524} C_DIS
LIN {X -51.5442,Y 110.7906,Z 131,A 110.4054,B 24.9439,C -1.7302,E1 24.9338,E2 335.7913} C_DIS
LIN {X -47.9769,Y 112.3824,Z 131,A 108.5193,B 24.9439,C -1.7304,E1 24.9386,E2 337.6812} C_DIS
LIN {X -42.8676,Y 114.4289,Z 131,A 105.7383,B 24.9442,C -1.7251,E1 24.9459,E2 340.4809} C_DIS
LIN {X -37.5494,Y 116.2825,Z 131,A 103.2879,B 24.9435,C -1.7368,E1 24.9523,E2 342.908} C_DIS
LIN {X -33.5625,Y 117.495,Z 131,A 101.3205,B 24.9434,C -1.7384,E1 24.9576,E2 344.8749} C_DIS
LIN {X -29.6414,Y 118.5448,Z 131,A 99.4806,B 24.9431,C -1.7432,E1 24.9625,E2 346.7062} C_DIS
LIN {X -26.015,Y 119.3927,Z 131,A 97.3734,B 24.944,C -1.7285,E1 24.9684,E2 348.8509} C_DIS
LIN {X -22.5279,Y 120.1001,Z 131,A 95.7049,B 24.944,C -1.7298,E1 24.973,E2 350.518} C_DIS
LIN {X -19.0419,Y 120.7022,Z 131,A 94.5659,B 24.9423,C -1.7545,E1 24.9759,E2 351.5995} C_DIS
LIN {X -16.1978,Y 121.116,Z 131,A 93.032,B 24.9428,C -1.7469,E1 24.9802,E2 353.1526} C_DIS
LIN {X -9.2558,Y 121.8433,Z 131,A 89.8355,B 24.9425,C -1.7521,E1 24.9891,E2 356.3386} C_DIS
LIN {X -3.3256,Y 122.1498,Z 131,A 86.9808,B 24.9426,C -1.7498,E1 24.9971,E2 359.1995} C_DIS
LIN {X 0.596,Y 122.1926,Z 131,A 85.0936,B 24.9427,C -1.748,E1 25.0024,E2 361.0909} C_DIS
LIN {X 5.0218,Y 122.0909,Z 131,A 82.6934,B 24.9437,C -1.7333,E1 25.0091,E2 363.5254} C_DIS
LIN {X 8.6418,Y 121.8883,Z 131,A 81.2971,B 24.9428,C -1.7472,E1 25.0129,E2 364.8881} C_DIS
LIN {X 12.7594,Y 121.5261,Z 131,A 79.4147,B 24.9426,C -1.7495,E1 25.0182,E2 366.7637} C_DIS
LIN {X 16.5486,Y 121.069,Z 131,A 77.0801,B 24.9443,C -1.7239,E1 25.0248,E2 369.1571} C_DIS
LIN {X 20.994,Y 120.3778,Z 131,A 74.8138,B 24.9448,C -1.716,E1 25.0311,E2 371.4399} C_DIS
LIN {X 26.1072,Y 119.3725,Z 131,A 73.2931,B 24.9421,C -1.7576,E1 25.035,E2 372.86} C_DIS
LIN {X 29.0484,Y 118.6917,Z 131,A 71.6903,B 24.9427,C -1.748,E1 25.0394,E2 374.4832} C_DIS
LIN {X 31.8521,Y 117.9699,Z 131,A 70.3089,B 24.9429,C -1.746,E1 25.0431,E2 375.8672} C_DIS
LIN {X 35.3846,Y 116.9598,Z 131,A 68.5419,B 24.9431,C -1.7427,E1 25.0478,E2 377.6391} C_DIS
LIN {X 39.3255,Y 115.6932,Z 131,A 66.6122,B 24.9431,C -1.7416,E1 25.0529,E2 379.5677} C_DIS
LIN {X 43.2035,Y 114.3016,Z 131,A 64.7389,B 24.9431,C -1.7425,E1 25.0578,E2 381.4347} C_DIS
LIN {X 48.6888,Y 112.0751,Z 131,A 61.9343,B 24.9434,C -1.7382,E1 25.0651,E2 384.2432} C_DIS
LIN {X 54.0871,Y 109.5728,Z 131,A 59.4149,B 24.9428,C -1.7476,E1 25.0714,E2 386.7337} C_DIS
LIN {X 58.1048,Y 107.4962,Z 131,A 57.0257,B 24.9438,C -1.732,E1 25.0774,E2 389.1532} C_DIS
LIN {X 61.474,Y 105.6051,Z 131,A 54.8427,B 24.9451,C -1.7117,E1 25.0827,E2 391.3777} C_DIS
LIN {X 64.771,Y 103.6158,Z 131,A 53.4326,B 24.9441,C -1.7277,E1 25.086,E2 392.7454} C_DIS
LIN {X 69.9625,Y 100.1834,Z 131,A 50.8789,B 24.9432,C -1.7404,E1 25.0919,E2 395.2606} C_DIS
LIN {X 73.5717,Y 97.5637,Z 131,A 48.4121,B 24.9446,C -1.7186,E1 25.0975,E2 397.7702} C_DIS
LIN {X 76.9284,Y 94.9398,Z 131,A 46.4452,B 24.9448,C -1.7163,E1 25.1018,E2 399.7352} C_DIS
LIN {X 79.9829,Y 92.381,Z 131,A 44.3075,B 24.9459,C -1.6996,E1 25.1064,E2 401.9039} C_DIS
LIN {X 82.4635,Y 90.1734,Z 131,A 43.0154,B 24.9453,C -1.7092,E1 25.109,E2 403.1681} C_DIS
LIN {X 85.5068,Y 87.2929,Z 131,A 41.0725,B 24.9455,C -1.7061,E1 25.1129,E2 405.1103} C_DIS
LIN {X 88.065,Y 84.7107,Z 131,A 39.3649,B 24.9457,C -1.7022,E1 25.1162,E2 406.8198} C_DIS
LIN {X 90.988,Y 81.563,Z 131,A 37.3957,B 24.9459,C -1.6998,E1 25.1199,E2 408.7859} C_DIS
LIN {X 93.7169,Y 78.4132,Z 131,A 35.4168,B 24.9462,C -1.694,E1 25.1235,E2 410.7696} C_DIS
LIN {X 96.3908,Y 75.1032,Z 131,A 33.4131,B 24.9466,C -1.6887,E1 25.127,E2 412.7764} C_DIS
LIN {X 98.8989,Y 71.7667,Z 131,A 31.4657,B 24.9468,C -1.6843,E1 25.1302,E2 414.7249} C_DIS
LIN {X 102.2758,Y 66.8674,Z 131,A 28.6824,B 24.9473,C -1.6773,E1 25.1346,E2 417.5108} C_DIS
LIN {X 106.3818,Y 60.1213,Z 131,A 24.9827,B 24.9479,C -1.6674,E1 25.1399,E2 421.2148} C_DIS
LIN {X 108.463,Y 56.2796,Z 131,A 22.9665,B 24.9482,C -1.6633,E1 25.1425,E2 423.2301} C_DIS
LIN {X 110.8928,Y 51.325,Z 131,A 20.6591,B 24.9478,C -1.6698,E1 25.1453,E2 425.5098} C_DIS
LIN {X 112.1024,Y 48.6259,Z 131,A 18.1564,B 24.9514,C -1.6108,E1 25.1482,E2 428.138} C_DIS
LIN {X 114.4764,Y 42.741,Z 131,A 16.0502,B 24.9493,C -1.6446,E1 25.1502,E2 430.1527} C_DIS
LIN {X 115.9167,Y 38.6638,Z 131,A 14.072,B 24.9495,C -1.6409,E1 25.152,E2 432.1285} C_DIS
LIN {X 117.1786,Y 34.6495,Z 131,A 12.146,B 24.9498,C -1.6372,E1 25.1536,E2 434.0522} C_DIS
LIN {X 118.282,Y 30.6718,Z 131,A 10.2401,B 24.95,C -1.6327,E1 25.155,E2 435.9579} C_DIS
LIN {X 120.0151,Y 22.9737,Z 131,A 6.9079,B 24.9496,C -1.6394,E1 25.157,E2 439.255} C_DIS
LIN {X 121.1687,Y 15.8021,Z 131,A 2.7835,B 24.9525,C -1.5925,E1 25.1588,E2 443.4656} C_DIS
LIN {X 121.5953,Y 12.0891,Z 131,A 1.644,B 24.951,C -1.6174,E1 25.1591,E2 444.5396} C_DIS
LIN {X 121.8412,Y 9.2839,Z 131,A 0.0741,B 24.952,C -1.6006,E1 25.1594,E2 446.1398} C_DIS
LIN {X 122.136,Y 3.7688,Z 131,A -2.7541,B 24.9532,C -1.5803,E1 25.1598,E2 448.9991} C_DIS
LIN {X 122.1933,Y 0.4456,Z 131,A -3.8555,B 24.9522,C -1.598,E1 25.1598,E2 450.0521} C_DIS
LIN {X 122.1648,Y -2.6898,Z 131,A -5.8733,B 24.9541,C -1.5658,E1 25.1597,E2 452.1339} C_DIS
LIN {X 122.0177,Y -6.5782,Z 131,A -7.2953,B 24.9532,C -1.5799,E1 25.1595,E2 453.5142} C_DIS
LIN {X 121.5757,Y -12.2875,Z 131,A -9.862,B 24.9534,C -1.577,E1 25.1589,E2 456.0725} C_DIS
LIN {X 121.1918,Y -15.6245,Z 131,A -11.5546,B 24.9541,C -1.5659,E1 25.1583,E2 457.7812} C_DIS
LIN {X 120.5582,Y -19.9333,Z 131,A -13.8537,B 24.9552,C -1.5464,E1 25.1573,E2 460.1128} C_DIS
LIN {X 119.9558,Y -23.2838,Z 131,A -15.0271,B 24.9543,C -1.5624,E1 25.1567,E2 461.2417} C_DIS
LIN {X 119.2556,Y -26.6402,Z 131,A -17.0598,B 24.9558,C -1.5359,E1 25.1555,E2 463.325} C_DIS
LIN {X 118.459,Y -29.9778,Z 131,A -18.4425,B 24.9555,C -1.542,E1 25.1545,E2 464.6854} C_DIS
LIN {X 117.228,Y -34.4832,Z 131,A -20.4305,B 24.9553,C -1.545,E1 25.153,E2 466.6548} C_DIS
LIN {X 116.1571,Y -37.9342,Z 131,A -22.2327,B 24.9559,C -1.5342,E1 25.1515,E2 468.4723} C_DIS
LIN {X 113.8512,Y -44.3769,Z 131,A -25.0131,B 24.9552,C -1.5456,E1 25.1489,E2 471.2103} C_DIS
LIN {X 110.7556,Y -51.6193,Z 131,A -28.6398,B 24.9557,C -1.5374,E1 25.1449,E2 474.8364} C_DIS
LIN {X 108.7267,Y -55.7662,Z 131,A -31.2278,B 24.9573,C -1.5096,E1 25.1416,E2 477.4761} C_DIS
LIN {X 106.5733,Y -59.7788,Z 131,A -33.1342,B 24.957,C -1.5147,E1 25.1391,E2 479.3605} C_DIS
LIN {X 105.0485,Y -62.4202,Z 131,A -35.1286,B 24.9588,C -1.4824,E1 25.1362,E2 481.4209} C_DIS
LIN {X 103.0193,Y -65.7162,Z 131,A -36.3164,B 24.9574,C -1.5083,E1 25.1345,E2 482.5416} C_DIS
LIN {X 99.8633,Y -70.4185,Z 131,A -39.1624,B 24.9583,C -1.4912,E1 25.13,E2 485.4137} C_DIS
LIN {X 98.1722,Y -72.7577,Z 131,A -41.095,B 24.9601,C -1.4588,E1 25.1267,E2 487.4135} C_DIS
LIN {X 95.31,Y -76.4688,Z 131,A -42.5206,B 24.9584,C -1.491,E1 25.1244,E2 488.7565} C_DIS
LIN {X 93.3187,Y -78.8864,Z 131,A -44.1668,B 24.9591,C -1.4783,E1 25.1214,E2 490.4252} C_DIS
LIN {X 89.5807,Y -83.107,Z 131,A -46.9971,B 24.9599,C -1.4622,E1 25.116,E2 493.2808} C_DIS
LIN {X 86.746,Y -86.0624,Z 131,A -48.6723,B 24.9595,C -1.4695,E1 25.1128,E2 494.9316} C_DIS
LIN {X 84.0167,Y -88.7278,Z 131,A -50.4748,B 24.9598,C -1.4645,E1 25.1092,E2 496.7385} C_DIS
LIN {X 80.6489,Y -91.7998,Z 131,A -52.8717,B 24.9608,C -1.4467,E1 25.1041,E2 499.1679} C_DIS
LIN {X 77.5113,Y -94.4646,Z 131,A -54.5574,B 24.9604,C -1.4543,E1 25.1006,E2 500.8292} C_DIS
LIN {X 74.5012,Y -96.8552,Z 131,A -56.2593,B 24.9604,C -1.4553,E1 25.0968,E2 502.5225} C_DIS
LIN {X 71.1835,Y -99.3192,Z 131,A -58.3842,B 24.961,C -1.442,E1 25.092,E2 504.6712} C_DIS
LIN {X 67.9155,Y -101.5828,Z 131,A -60.0685,B 24.9608,C -1.447,E1 25.0881,E2 506.3381} C_DIS
LIN {X 62.5339,Y -104.9807,Z 131,A -63.4259,B 24.9621,C -1.423,E1 25.0801,E2 509.7413} C_DIS
LIN {X 59.448,Y -106.7583,Z 131,A -64.7755,B 24.9614,C -1.4356,E1 25.0769,E2 511.0573} C_DIS
LIN {X 56.1626,Y -108.5238,Z 131,A -66.5542,B 24.9616,C -1.4311,E1 25.0724,E2 512.8416} C_DIS
LIN {X 52.128,Y -110.5184,Z 131,A -68.9852,B 24.9626,C -1.4122,E1 25.0662,E2 515.311} C_DIS
LIN {X 48.7154,Y -112.0634,Z 131,A -70.6204,B 24.9625,C -1.4153,E1 25.0621,E2 516.9347} C_DIS
LIN {X 45.6721,Y -113.3383,Z 131,A -71.8486,B 24.9618,C -1.4285,E1 25.059,E2 518.129} C_DIS
LIN {X 41.9121,Y -114.7822,Z 131,A -73.8084,B 24.9621,C -1.4224,E1 25.0538,E2 520.099} C_DIS
LIN {X 36.8395,Y -116.509,Z 131,A -75.9447,B 24.9613,C -1.4375,E1 25.0483,E2 522.1956} C_DIS
LIN {X 32.298,Y -117.8494,Z 131,A -78.5445,B 24.9624,C -1.4166,E1 25.0412,E2 524.8403} C_DIS
LIN {X 26.5653,Y -119.272,Z 131,A -81.1822,B 24.9622,C -1.4202,E1 25.0341,E2 527.4657} C_DIS
LIN {X 22.7919,Y -120.0497,Z 131,A -83.4059,B 24.9633,C -1.3988,E1 25.0278,E2 529.7375} C_DIS
LIN {X 19.1919,Y -120.6784,Z 131,A -84.7849,B 24.9626,C -1.4134,E1 25.0241,E2 531.0806} C_DIS
LIN {X 13.7699,Y -121.416,Z 131,A -87.1299,B 24.9621,C -1.4222,E1 25.0177,E2 533.4027} C_DIS
LIN {X 10.8592,Y -121.7111,Z 131,A -88.667,B 24.9626,C -1.4136,E1 25.0134,E2 534.9592} C_DIS
LIN {X 5.8258,Y -122.0559,Z 131,A -91.017,B 24.9626,C -1.4133,E1 25.0068,E2 537.309} C_DIS
LIN {X 0.8751,Y -122.1912,Z 131,A -93.0926,B 24.962,C -1.4242,E1 25.0011,E2 539.3583} C_DIS
Enddeposition()
LIN {X 0.8751,Y -122.1912,Z 131,A -93.0926,B 24.962,C -1.4242,E1 25.0011,E2 539.3583} C_DIS
Startdeposition()
$VEL.CP = VEL_PRINT
LIN {X 5.052,Y -121.2482,Z 131,A -90.8396,B 24.9605,C -1.4528,E1 25.0076,E2 537.038} C_DIS
LIN {X 10.6575,Y -120.8849,Z 131,A -87.9219,B 24.9597,C -1.4666,E1 25.0158,E2 534.089} C_DIS
LIN {X 18.8375,Y -119.8832,Z 131,A -83.3133,B 24.9576,C -1.5039,E1 25.0288,E2 529.3961} C_DIS
LIN {X 24.3281,Y -118.8906,Z 131,A -81.3952,B 24.9594,C -1.4714,E1 25.0338,E2 527.5573} C_DIS
LIN {X 26.9784,Y -118.3167,Z 131,A -79.7935,B 24.9585,C -1.4882,E1 25.0383,E2 525.918} C_DIS
LIN {X 30.6336,Y -117.4237,Z 131,A -78.354,B 24.9593,C -1.4737,E1 25.0421,E2 524.515} C_DIS
LIN {X 34.6259,Y -116.3086,Z 131,A -76.4299,B 24.9593,C -1.4743,E1 25.0472,E2 522.5927} C_DIS
LIN {X 37.4028,Y -115.4464,Z 131,A -74.0191,B 24.9563,C -1.5269,E1 25.054,E2 520.0622} C_DIS
LIN {X 43.9472,Y -113.1165,Z 131,A -71.9626,B 24.9594,C -1.4713,E1 25.059,E2 518.1417} C_DIS
Enddeposition()
END
